METHOD Praca : BOOL
VAR_INPUT
END_VAR
tonOdczekaj (PT := REAL_TO_TIME (stParametry.rOdczekaj));
fbNaped.Praca ();

SUPER^.Praca ();
END_METHOD

METHOD Resetowanie : BOOL
VAR_INPUT
END_VAR
tonOdczekaj.IN								:= FALSE;

SUPER^.Resetowanie ();
END_METHOD

END_FUNCTION_BLOCK

// ---- POUs/93 - Podzespol/POU/FB_Podzespol.TcPOU
//==================================================================================================
//								RJM Maszyny sp. z o.o.
//									13.05.2022
//	Obsluga przesuwacza na siłowniku 
//	Siłownik zabieraka plus siłownik przesuwający 
//	Cykl przesuwania: wysun zabierak -> przesun -> schowaj zabierak -> powrót  
// 	v1.0	|| TC v 3.1.4024.22		|| - pierwsza wersja
//==================================================================================================
FUNCTION_BLOCK FB_Podzespol IMPLEMENTS ITF_Podzespol
VAR_INPUT
	//Parametry
END_VAR
VAR_OUTPUT
END_VAR
VAR
	//Elementy wejsciowe i wykonawcze
	bBazuj									: BOOL;
	bBazowanie								: BOOL;
	bCyklBazowaniaSkonczony					: BOOL;
	bPierwszePrzejscieBazowanie				: BOOL;
	iKrokBazowania							: INT :=0;

	bWykonajCyklPracy						: BOOL;
	bCyklPracy								: BOOL;
	bCyklPracySkonczony						: BOOL;
	bPierwszePrzejsciePracy					: BOOL;
	iKrokPracy								: INT := 0;

	bReset									: BOOL;
END_VAR

PROPERTY Bazowanie : BOOL
GET
Bazowanie									:= bBazowanie;
END_GET
END_PROPERTY

PROPERTY Bazuj : BOOL
SET
bBazuj										:= Bazuj;
END_SET
END_PROPERTY

METHOD CyklBazowania_Praca : BOOL
VAR_INPUT
END_VAR
END_METHOD

PROPERTY CyklPracy : BOOL
GET
CyklPracy								:= bCyklPracy;
END_GET
END_PROPERTY

METHOD CyklPracy_Praca : BOOL
VAR_INPUT
END_VAR
END_METHOD

PROPERTY CyklPracySkonczony : BOOL
GET
CyklPracySkonczony					:= bCyklPracySkonczony;
END_GET
END_PROPERTY

PROPERTY Pozycja0 : BOOL
GET
END_GET
END_PROPERTY

METHOD Praca : BOOL
VAR_INPUT
END_VAR
//---------------Resetowanie zmiennych
	IF (bReset) THEN
		Resetowanie ();
	END_IF
//---------------Resetowanie zmiennych
//---------------Bazowanie siłowników - powrót do poczatku
	IF (bBazuj) THEN
		bPierwszePrzejscieBazowanie				:= FALSE;
		bBazowanie								:= TRUE;
		bBazuj									:= FALSE;
	END_IF
	IF (bBazowanie) THEN
		bBazowanie								:= CyklBazowania_Praca ();
	END_IF
//---------------Bazowanie siłowników - powrót do poczatku
//---------------Cykl przesuwnaia - koniec gora dol poczatek
	IF (bWykonajCyklPracy) THEN
		bCyklPracy						:= TRUE;
	END_IF
	IF (bCyklPracy) THEN
		bCyklPracy						:= CyklPracy_Praca ();
	END_IF
//---------------Cykl przesuwnaia - koniec gora dol poczatek
END_METHOD

METHOD Resetowanie : BOOL
VAR_INPUT
END_VAR
bWykonajCyklPracy							:= FALSE;
bCyklPracy									:= FALSE;
bCyklPracySkonczony							:= FALSE;
bBazuj										:= false;
bBazowanie									:= false;
bCyklBazowaniaSkonczony						:= FALSE;
bPierwszePrzejscieBazowanie					:= FALSE;
bPierwszePrzejsciePracy						:= FALSE;
iKrokBazowania								:= 0;
iKrokPracy									:= 0;



bReset										:= FALSE;
END_METHOD

PROPERTY Resetuj : BOOL
SET
bReset										:=Resetuj;
END_SET
END_PROPERTY

PROPERTY WykonajCyklPracy : BOOL
SET
bWykonajCyklPracy						:= WykonajCyklPracy;
END_SET
END_PROPERTY

END_FUNCTION_BLOCK

// ---- POUs/03 - Ciecie/POU/FB_Ciecie_Komunikacja.TcPOU
FUNCTION_BLOCK FB_Ciecie_Komunikacja EXTENDS FB_LogowanieBledow_ElementZlozony
VAR_INPUT
END_VAR
VAR_OUTPUT
END_VAR
VAR
END_VAR

METHOD DefinicjaTabeliZdarzen_1031_Niemiecki : BOOL
VAR_INPUT
	arrTablicaDefinicjiZdarzenOpis			: REFERENCE TO ARRAY [1..GVL_LogowanieBledow_Stale.MAX_ILOSC_ZDARZEN] OF DUT_LogowanieBledow_ZdarzenieOpis;

END_VAR
//arrTablicaDefinicjiZdarzenOpis [iStartId+0].sOpis	:= 'DE - TESTOWA WIADOMOSC';
END_METHOD

METHOD DefinicjaTabeliZdarzen_1033_Angielski : BOOL
VAR_INPUT
	arrTablicaDefinicjiZdarzenOpis			: REFERENCE TO ARRAY [1..GVL_LogowanieBledow_Stale.MAX_ILOSC_ZDARZEN] OF DUT_LogowanieBledow_ZdarzenieOpis;

END_VAR
//arrTablicaDefinicjiZdarzenOpis [iStartId+0].sOpis	:= 'EN - TESTOWA WIADOMOSC';
END_METHOD

METHOD DefinicjaTabeliZdarzen_1045_Polski : BOOL
VAR_INPUT
	arrTablicaDefinicjiZdarzenOpis			: REFERENCE TO ARRAY [1..GVL_LogowanieBledow_Stale.MAX_ILOSC_ZDARZEN] OF DUT_LogowanieBledow_ZdarzenieOpis;

END_VAR
//arrTablicaDefinicjiZdarzenOpis [iStartId+0].sOpis	:= 'PL - TESTOWA WIADOMOSC';
END_METHOD

METHOD DefinicjaTabeliZdarzen_Ogolna : BOOL
VAR_INPUT
	arrTablicaDefinicjiZdarzen				: REFERENCE TO ARRAY [1..GVL_LogowanieBledow_Stale.MAX_ILOSC_ZDARZEN] OF DUT_LogowanieBledow_Zdarzenie;
	arrTablicaDefinicjiZdarzenOpis			: REFERENCE TO ARRAY [1..GVL_LogowanieBledow_Stale.MAX_ILOSC_ZDARZEN] OF DUT_LogowanieBledow_ZdarzenieOpis;
	arrTablicaDefinicjiZdarzenStan			: REFERENCE TO ARRAY [1..GVL_LogowanieBledow_Stale.MAX_ILOSC_ZDARZEN] OF DUT_LogowanieBledow_ZdarzenieStan;

	iIdZdarzenia							: REFERENCE TO INT;
	iNrPodzespolu							: INT := 0;
	iNrPodelementu							: INT := 0;
	iNrElementu								: INT := 0;
END_VAR
(*
//testowy blad
	iIdZdarzenia												:= iIdZdarzenia + 1;
	arrTablicaDefinicjiZdarzen [iIdZdarzenia].iIdZdarzenia		:= iIdZdarzenia;
	arrTablicaDefinicjiZdarzen [iIdZdarzenia].byRodzajZdarzenia	:= 3;
	arrTablicaDefinicjiZdarzen [iIdZdarzenia].sKodBledu			:= '0001';
	arrTablicaDefinicjiZdarzen [iIdZdarzenia].sNrKomponentu		:= GenerujNrKomponentu (iNrPodzespolu := iNrPodzespolu, iNrPodelementu := iNrPodelementu, iNrElementu := iNrElementu); 
	arrTablicaDefinicjiZdarzenOpis [iIdZdarzenia].iIdZdarzenia 	:= iIdZdarzenia;
	arrTablicaDefinicjiZdarzenStan [iIdZdarzenia].iIdZdarzenia 	:= iIdZdarzenia;
	arrTablicaDefinicjiZdarzenStan [iIdZdarzenia].bAktywne		:= FALSE;
	*)
END_METHOD

END_FUNCTION_BLOCK

// ---- POUs/95 - Logowanie bledow/POU/FB_LogowanieBledow_ElementZlozony.TcPOU
//==================================================================================================
//								RJM Maszyny sp. z o.o.
//									14.06.2022
//	FB posredniczący pomiędzy FB a logerem alarmów  rozszerzenie dla elementów złożonych
// 	v1.0	|| TC v 3.1.4024.22		|| - pierwsza wersja
//==================================================================================================
FUNCTION_BLOCK FB_LogowanieBledow_ElementZlozony EXTENDS FB_LogowanieBledow_ElementWykonawczy
VAR_INPUT
	
END_VAR
VAR_OUTPUT
END_VAR
VAR
	arrElementyWykonawcze 					: ARRAY [1..GVL_LogowanieBledow_Stale.MAX_ILOSC_ELEMENTOW_NA_PODZESPOL] OF ITF_LogowanieBledow_ElementWykonawczy;
	iIloscPodlementow						: INT;
END_VAR

METHOD DefinicjaTabeliZdarzen_1031_Niemiecki : BOOL
VAR_INPUT
	arrTablicaDefinicjiZdarzenOpis			: REFERENCE TO ARRAY [1..GVL_LogowanieBledow_Stale.MAX_ILOSC_ZDARZEN] OF DUT_LogowanieBledow_ZdarzenieOpis;

END_VAR
END_METHOD

METHOD DefinicjaTabeliZdarzen_1033_Angielski : BOOL
VAR_INPUT
	arrTablicaDefinicjiZdarzenOpis			: REFERENCE TO ARRAY [1..GVL_LogowanieBledow_Stale.MAX_ILOSC_ZDARZEN] OF DUT_LogowanieBledow_ZdarzenieOpis;

END_VAR
END_METHOD

METHOD DefinicjaTabeliZdarzen_1045_Polski : BOOL
VAR_INPUT
	arrTablicaDefinicjiZdarzenOpis			: REFERENCE TO ARRAY [1..GVL_LogowanieBledow_Stale.MAX_ILOSC_ZDARZEN] OF DUT_LogowanieBledow_ZdarzenieOpis;

END_VAR
END_METHOD

METHOD DefinicjaTabeliZdarzen_Ogolna : BOOL
VAR_INPUT
	arrTablicaDefinicjiZdarzen				: REFERENCE TO ARRAY [1..GVL_LogowanieBledow_Stale.MAX_ILOSC_ZDARZEN] OF DUT_LogowanieBledow_Zdarzenie;
	arrTablicaDefinicjiZdarzenOpis			: REFERENCE TO ARRAY [1..GVL_LogowanieBledow_Stale.MAX_ILOSC_ZDARZEN] OF DUT_LogowanieBledow_ZdarzenieOpis;
	arrTablicaDefinicjiZdarzenStan			: REFERENCE TO ARRAY [1..GVL_LogowanieBledow_Stale.MAX_ILOSC_ZDARZEN] OF DUT_LogowanieBledow_ZdarzenieStan;

	iIdZdarzenia							: REFERENCE TO INT;
	iNrPodzespolu							: INT := 0;
	iNrPodelementu							: INT := 0;
	iNrElementu								: INT := 0;
END_VAR
END_METHOD

METHOD FB_init : BOOL
VAR_INPUT
	bInitRetains : BOOL; // if TRUE, the retain variables are initialized (warm start / cold start)
	bInCopyCode : BOOL;  // if TRUE, the instance afterwards gets moved into the copy code (online change)
	arrElementyWykonawcze 					: ARRAY [1..10] OF ITF_LogowanieBledow_ElementWykonawczy;
	iIloscPodlementow						: INT;
END_VAR
THIS^.arrElementyWykonawcze					:= arrElementyWykonawcze;
THIS^.iIloscPodlementow						:= iIloscPodlementow;
END_METHOD

METHOD ZwrocTabliceDefinicji : BOOL
VAR_INPUT
	arrTablicaDefinicjiZdarzen				: REFERENCE TO ARRAY [1..GVL_LogowanieBledow_Stale.MAX_ILOSC_ZDARZEN] OF DUT_LogowanieBledow_Zdarzenie;
	arrTablicaDefinicjiZdarzenOpis			: REFERENCE TO ARRAY [1..GVL_LogowanieBledow_Stale.MAX_ILOSC_ZDARZEN] OF DUT_LogowanieBledow_ZdarzenieOpis;
	arrTablicaDefinicjiZdarzenStan			: REFERENCE TO ARRAY [1..GVL_LogowanieBledow_Stale.MAX_ILOSC_ZDARZEN] OF DUT_LogowanieBledow_ZdarzenieStan;
	
	iIdZdarzenia							: REFERENCE TO INT;
	iNrPodzespolu							: INT;
	iNrPodelementu							: INT;
	iNrElementu								: INT;
	iJezykId								: INT;
END_VAR
VAR
	iI: INT;
END_VAR
//Zwrócenie definicji zdarzen dla głównego elementu 
SUPER^.ZwrocTabliceDefinicji (	arrTablicaDefinicjiZdarzen := arrTablicaDefinicjiZdarzen,
								arrTablicaDefinicjiZdarzenOpis := arrTablicaDefinicjiZdarzenOpis,
								arrTablicaDefinicjiZdarzenStan := arrTablicaDefinicjiZdarzenStan,
								iIdZdarzenia := iIdZdarzenia,
								iNrPodzespolu := iNrPodzespolu, 
								iNrPodelementu := iNrPodelementu,
								iNrElementu := 1, 
								iJezykId := iJezykID);
//zwrócenie tablicy definicji dla podelementów

	FOR iI := 1 TO iIloscPodlementow DO 
		arrElementyWykonawcze [iI].ZwrocTabliceDefinicji (	arrTablicaDefinicjiZdarzen := arrTablicaDefinicjiZdarzen,
															arrTablicaDefinicjiZdarzenOpis := arrTablicaDefinicjiZdarzenOpis,
															arrTablicaDefinicjiZdarzenStan := arrTablicaDefinicjiZdarzenStan,
															iIdZdarzenia := iIdZdarzenia, 
															iNrPodzespolu := iNrPodzespolu, 
															iNrPodelementu := iNrPodelementu,
															iNrElementu := iI+1, 
															iJezykId := iJezykID);
	END_FOR
END_METHOD

METHOD ZwrocTabliceStanu : BOOL
VAR_INPUT
	arrTablicaDefinicjiZdarzenStan			: REFERENCE TO ARRAY [1..GVL_LogowanieBledow_Stale.MAX_ILOSC_ZDARZEN] OF DUT_LogowanieBledow_ZdarzenieStan;
END_VAR

VAR
	iI										: INT;
	iJ										: INT;
END_VAR
SUPER^.ZwrocTabliceStanu (arrTablicaDefinicjiZdarzenStan := arrTablicaDefinicjiZdarzenStan);

FOR iJ := 1 TO iIloscPodlementow DO
	arrElementyWykonawcze [iJ].ZwrocTabliceStanu (arrTablicaDefinicjiZdarzenStan := arrTablicaDefinicjiZdarzenStan);
END_FOR
END_METHOD

END_FUNCTION_BLOCK

// ---- POUs/02 - Przesuwacz Na Silowniku/POU/FB_PrzesuwaczNaSilowniku.TcPOU
//==================================================================================================
//								RJM Maszyny sp. z o.o.
//									13.05.2022
//	Obsluga przesuwacza na siłowniku 
//	Siłownik zabieraka plus siłownik przesuwający 
//	Cykl przesuwania: wysun zabierak -> przesun -> schowaj zabierak -> powrót  
// 	v1.0	|| TC v 3.1.4024.22		|| - pierwsza wersja
//==================================================================================================
FUNCTION_BLOCK FB_PrzesuwaczNaSilowniku EXTENDS FB_Podzespol
VAR_INPUT
	stParametry								: DUT_PrzesuwaczNaSilowniku_Parametry;
END_VAR
VAR_OUTPUT
END_VAR
VAR
	bCzujnik0Zabieraka						: ITF_Czujnik;
	bCzujnikMaxZabieraka					: ITF_Czujnik;
	fbElektrozaworZabieraka					: ITF_Elektozawor;
	bCzujnik0Przesuwacza					: ITF_Czujnik;
	bCzujnikMaxPrzesuwacza					: ITF_Czujnik;
	fbElektrozaworPrzesuwacza				: ITF_Elektozawor;
	fbZabierak								: FB_Silownik_Kontrola (	fbCzujnikPozycja0 			:= GVL_Wejscia_IO.bCzujnik0PW_Z, 
																		fbCzujnikPozycjaMax 		:= GVL_Wejscia_IO.bCzujnikMaxPW_Z,
																		fbElektrozawor 				:= GVL_Wyjscia_IO.fbElektrozaworPW_Z);
	fbPrzesuwanie							: FB_Silownik_Kontrola (	fbCzujnikPozycja0 			:= GVL_Wejscia_IO.bCzujnik0PW_N, 
																		fbCzujnikPozycjaMax 		:= GVL_Wejscia_IO.bCzujnikMaxPW_N,
																		fbElektrozawor 				:= GVL_Wyjscia_IO.fbElektrozaworPW_N);

	arrElementyWykonawcze 					: ARRAY [1..GVL_LogowanieBledow_Stale.MAX_ILOSC_ELEMENTOW_NA_PODZESPOL] OF ITF_LogowanieBledow_ElementWykonawczy := 
														[fbZabierak.fbLBKomunikacja, 
														fbPrzesuwanie.fbLBKomunikacja];
	fbLBKomunikacja							: FB_PrzesuwaczNaSilowniku_Komunikacja 
														(arrElementyWykonawcze := arrElementyWykonawcze,
														iIloscPodlementow := 2);

	tonChwilaPoDojechaniu					: TON;
END_VAR

METHOD CyklBazowania_Praca : BOOL
VAR_INPUT
END_VAR
IF (NOT bPierwszePrzejscieBazowanie) THEN
	bPierwszePrzejscieBazowanie				:= TRUE;
	bCyklBazowaniaSkonczony					:= FALSE;
	fbZabierak.PrzesunDoPoczatku			:= TRUE;
	iKrokBazowania							:= 1;
END_IF

CASE iKrokBazowania OF
	1	:
		IF (fbZabierak.NaPoczatku) THEN
			fbPrzesuwanie.PrzesunDoPoczatku	:= TRUE;
			iKrokBazowania					:= 10;
		END_IF
		CyklBazowania_Praca					:= TRUE;
	10	:
		IF (fbPrzesuwanie.NaPoczatku AND fbZabierak.NaPoczatku) THEN
			bPierwszePrzejscieBazowanie		:= FALSE;
			bCyklBazowaniaSkonczony			:= TRUE;
			CyklBazowania_Praca				:= FALSE;
			iKrokBazowania					:= 0;
		ELSE
			CyklBazowania_Praca				:= TRUE;
		END_IF
		
END_CASE
END_METHOD

METHOD CyklPracy_Praca : BOOL
VAR_INPUT
END_VAR
IF (NOT bPierwszePrzejsciePracy) THEN
	bPierwszePrzejsciePracy					:= TRUE;
	bCyklPracySkonczony						:= FALSE;
	fbZabierak.PrzesunDoKonca				:= TRUE;
	tonChwilaPoDojechaniu.IN				:= FALSE;
	iKrokPracy								:= 1;
END_IF

CASE iKrokPracy OF
	1	:
	IF (fbZabierak.NaKoncu) THEN
		fbPrzesuwanie.PrzesunDoKonca	:= TRUE;
		iKrokPracy							:= 10;
	END_IF
	CyklPracy_Praca							:= TRUE;
	10	:
	IF (fbPrzesuwanie.NaKoncu) THEN
		tonChwilaPoDojechaniu.IN			:= TRUE;
		iKrokPracy							:= 20;
	END_IF
	CyklPracy_Praca							:= TRUE;
	20	:
	IF (tonChwilaPoDojechaniu.Q) THEN
		tonChwilaPoDojechaniu.IN			:= FALSE;
		fbZabierak.PrzesunDoKonca			:= TRUE;
		iKrokPracy							:= 30;
	END_IF
	CyklPracy_Praca							:= TRUE;
	30	:
	IF (fbZabierak.NaPoczatku) THEN
		fbPrzesuwanie.PrzesunDoPoczatku	:= TRUE;
		iKrokPracy							:= 40;
	END_IF
	CyklPracy_Praca							:= TRUE;
	40	:
	IF (fbPrzesuwanie.NaPoczatku) THEN
		iKrokPracy							:= 50;
		bCyklPracySkonczony					:= TRUE;
	END_IF
	CyklPracy_Praca							:= TRUE;
	50	:
		iKrokPracy							:= 0;
		CyklPracy_Praca						:= FALSE;
END_CASE
END_METHOD

METHOD FB_init : BOOL
VAR_INPUT
	bInitRetains : BOOL; // if TRUE, the retain variables are initialized (warm start / cold start)
	bInCopyCode : BOOL;  // if TRUE, the instance afterwards gets moved into the copy code (online change)
	bCzujnik0Zabieraka						: ITF_Czujnik;
	bCzujnikMaxZabieraka					: ITF_Czujnik;
	fbElektrozaworZabieraka					: ITF_Elektozawor;
	bCzujnik0Przesuwacza					: ITF_Czujnik;
	bCzujnikMaxPrzesuwacza					: ITF_Czujnik;
	fbElektrozaworPrzesuwacza				: ITF_Elektozawor;
	
END_VAR

THIS^.bCzujnik0Zabieraka					:= bCzujnik0Zabieraka;			     
THIS^.bCzujnikMaxZabieraka					:= bCzujnikMaxZabieraka;		    
THIS^.fbElektrozaworZabieraka				:= fbElektrozaworZabieraka;		 
THIS^.bCzujnik0Przesuwacza					:= bCzujnik0Przesuwacza;		    
THIS^.bCzujnikMaxPrzesuwacza				:= bCzujnikMaxPrzesuwacza;		  
THIS^.fbElektrozaworPrzesuwacza				:= fbElektrozaworPrzesuwacza;

THIS^.fbZabierak.FB_init (FALSE, FALSE, bCzujnik0Zabieraka, bCzujnikMaxZabieraka, fbElektrozaworZabieraka);
THIS^.fbPrzesuwanie.FB_init (FALSE, FALSE, bCzujnik0Przesuwacza, bCzujnikMaxPrzesuwacza, fbElektrozaworPrzesuwacza);
END_METHOD

PROPERTY Pozycja0 : BOOL
GET
Pozycja0									:= fbZabierak.NaPoczatku AND fbPrzesuwanie.NaPoczatku;
END_GET
END_PROPERTY

METHOD Praca : BOOL
VAR_INPUT
END_VAR
tonChwilaPoDojechaniu (PT := REAL_TO_TIME (stParametry.rCzasNaKoncu));

fbZabierak.Praca ();
fbPrzesuwanie.Praca ();


SUPER^.Praca ();
END_METHOD

METHOD Resetowanie : BOOL
VAR_INPUT
END_VAR
tonChwilaPoDojechaniu.IN					:= FALSE;

SUPER^.Resetowanie ();
END_METHOD

END_FUNCTION_BLOCK

// ---- POUs/01 - Elementy/Czujnik/POU/FB_Czujnik_NO.TcPOU
//==================================================================================================
//								RJM Maszyny sp. z o.o.
//									04.06.2022
//	Obsługa czujnika  NO
// 	v1.0	|| TC v 3.1.4024.22		|| - pierwsza wersja
//==================================================================================================
FUNCTION_BLOCK FB_Czujnik_NO IMPLEMENTS ITF_Czujnik
VAR_INPUT
	bSymulacja								: BOOL;
END_VAR
VAR
	bWejscie						AT %I*	: BOOL;
END_VAR

//==================================================================================================
//								RJM Maszyny sp. z o.o.
//									13.05.2022
//	Informacja czy czujnik jest zadziałany 
// 	v1.0	|| TC v 3.1.4024.22		|| - pierwsza wersja
//==================================================================================================
PROPERTY CzyZadzialany : BOOL
GET
CzyZadzialany								:= bWejscie;
END_GET
END_PROPERTY

END_FUNCTION_BLOCK

// ---- POUs/01 - Elementy/Elektrozawór/POU/FB_Elektrozawor_5na2_2Cewki.TcPOU
//==================================================================================================
//								RJM Maszyny sp. z o.o.
//									04.06.2022
//	Sterowanie elektrozaworem  - 5 na 2 z dwiema cewkami
// 	v1.0	|| TC v 3.1.4024.22		|| - pierwsza wersja
//==================================================================================================
FUNCTION_BLOCK FB_Elektrozawor_5na2_2Cewki IMPLEMENTS ITF_Elektozawor
VAR
	bCewkaA							AT %Q*	: BOOL;		//Cewka sterująca wyjściem 2 - 0 do MAX
	bCewkaB							AT %Q*	: BOOL;		//Cewka sterująca wyjściem 4 - MAX do 0
END_VAR

(*==================================================================================================
								RJM Maszyny sp. z o.o.
									04.06.2022
	Sterowanie cewkami elektrozaworu 
 	v1.0	|| TC v 3.1.4024.22		|| - pierwsza wersja
==================================================================================================*)
METHOD Steruj : BOOL
VAR_INPUT
	bKierunekWstrone0						: BOOL;
	bKierunekWStroneMax						: BOOL;
END_VAR
IF (bKierunekWStroneMax AND NOT bCewkaA) THEN
	bCewkaA									:= TRUE;
END_IF
IF  (bKierunekWstrone0 AND bCewkaA) THEN
	bCewkaA									:= FALSE;
END_IF

IF (bKierunekWstrone0 AND NOT bCewkaB) THEN
	bCewkaB									:= TRUE;
END_IF
IF  (bKierunekWStroneMax AND bCewkaB) THEN
	bCewkaB									:= FALSE;
END_IF
END_METHOD

END_FUNCTION_BLOCK

// ---- POUs/90 - Stan Maszyny/POU/FB_StanMaszyny.TcPOU
//==================================================================================================
//								RJM Maszyny sp. z o.o.
//									13.05.2022
//	Sterowanie pracą maszyny i jej trybami  
// 	v1.0	|| TC v 3.1.4024.29		|| - pierwsza wersja
//==================================================================================================
FUNCTION_BLOCK FB_StanMaszyny
VAR_INPUT
	bStart                                  : BOOL;
	bStop                                   : bool;
	bReset                                  : bool;
	bAbort                                  : bool;
	bClear                                  : bool;
	bHold                                   : bool;
	bUnHold                                 : bool;
	bSuspend                                : bool;
	bUnsuspend								: BOOL;
	eTryb									: E_PMLUnitMode;	//zadany tryb pracy
END_VAR
VAR_OUTPUT
END_VAR
VAR
	arrVisuStany							: ARRAY [0..17] OF DUT_StanMaszyny_VISU_Stan;
	arrVisuTryb								: ARRAY [0..9] of ARRAY [0..17] OF BOOL;
	eStan									: E_PMLState := E_PMLState.ABORTING;		//aktualny stan maszyny
	eTrybPracy								: E_PMLUnitMode := E_PMLUnitMode.MANUAL;	//aktualny tryb pracy
	
	arrPodzesoly							: ARRAY [1..GVL_StanMaszyny_Stale.MAX_LICZBA_PODZESPOLOW] OF ITF_StanMaszyny;
	iIloscDodanychPodzespolow				: INT;

	iAktualnyStan							: INT;
	iPoprzedniStan							: INT;
	iNumerTrybuPracy						: INT;
	iPoprzedniTrybPracy						: INT;

	bResetingSkonczone						: BOOL;
	bStoppingZakonczone						: BOOL;
	bAbortingZakonczone						: BOOL;
	bClearingZakonczone						: BOOL;
	bCompletingZakonczone					: BOOL;
	bHoldingZakonczone						: BOOL;
	bStartingZakonczone						: BOOL;
	bSuspendingZakonczone					: BOOL;
	bUnholdingZakonczone					: BOOL;
	bUnsuspendingZakonczone					: BOOL;	
	bInicjalizacja							: BOOL;
	bPierwszePrzejscieWOperacji				: BOOL;
	arrOperacjaWykonana						: ARRAY [1..GVL_StanMaszyny_Stale.MAX_LICZBA_PODZESPOLOW] OF BOOL;	//tablica zakonczenia zadanej operacji przez podzespoly
END_VAR

IF (NOT bInicjalizacja) THEN
	bInicjalizacja							:= TRUE;
	Inicjalizacja ();
END_IF



StanMaszyny ();

METHOD FB_init : BOOL
VAR_INPUT
	bInitRetains : BOOL; // if TRUE, the retain variables are initialized (warm start / cold start)
	bInCopyCode : BOOL;  // if TRUE, the instance afterwards gets moved into the copy code (online change)
	arrPodzesoly							: ARRAY [1..GVL_StanMaszyny_Stale.MAX_LICZBA_PODZESPOLOW] OF ITF_StanMaszyny;
	iIloscDodanychPodzespolow				: INT;
END_VAR
THIS^.arrPodzesoly								:= arrPodzesoly;
THIS^.iIloscDodanychPodzespolow					:= iIloscDodanychPodzespolow;
END_METHOD

//==================================================================================================
//								RJM Maszyny sp. z o.o.
//									13.05.2022
//	Iniecjalizacja tablicy potrzebnej do wyświetlania diagramu  
// 	v1.0	|| TC v 3.1.4024.29		|| - pierwsza wersja
//==================================================================================================
METHOD PRIVATE Inicjalizacja : BOOL
VAR_INPUT
END_VAR

VAR
	i,j: INT;
END_VAR


FOR j := 0 TO 9 DO
	FOR i := 0 TO 17 DO
		arrVisuStany [i].bAktywny				:= FALSE;
		CASE i OF
			0	:
				arrVisuStany [i].sNazwa			:= 'UNDEFINED';
				arrVisuStany [i].dwKolorTla		:= 16#FFFF0000;	//czerwony
			1	:             
				arrVisuStany [i].sNazwa			:= 'CLEARING';
				arrVisuStany [i].dwKolorTla		:= 16#FF00FF00;	//zielony
			2	:             
				arrVisuStany [i].sNazwa			:= 'STOPPED';
				arrVisuStany [i].dwKolorTla		:= 16#FFFFFF00;	//zolty
			3	:
				arrVisuStany [i].sNazwa			:= 'STARTING';
				arrVisuStany [i].dwKolorTla		:= 16#FF00FF00;
			4	:             
				arrVisuStany [i].sNazwa			:= 'IDLE';
				arrVisuStany [i].dwKolorTla		:= 16#FFFFFF00;
			5	:             
				arrVisuStany [i].sNazwa			:= 'SUSPENDED';
				arrVisuStany [i].dwKolorTla		:= 16#FFFFFF00;		
			6	:             
				arrVisuStany [i].sNazwa			:= 'EXECUTE';
				arrVisuStany [i].dwKolorTla		:= 16#FF0000FF;
			7	:             
				arrVisuStany [i].sNazwa			:= 'STOPPING';
				arrVisuStany [i].dwKolorTla		:= 16#FF00FF00;
			8	:             
				arrVisuStany [i].sNazwa			:= 'ABORTING';
				arrVisuStany [i].dwKolorTla		:= 16#FF00FF00;		
			9	:             
				arrVisuStany [i].sNazwa			:= 'ABORTED';
				arrVisuStany [i].dwKolorTla		:= 16#FFFFFF00;
			10	:             
				arrVisuStany [i].sNazwa			:= 'HOLDING';
				arrVisuStany [i].dwKolorTla		:= 16#FF00FF00;
			11	:             
				arrVisuStany [i].sNazwa			:= 'HELD';
				arrVisuStany [i].dwKolorTla		:= 16#FFFFFF00;	
			12	:             
				arrVisuStany [i].sNazwa			:= 'UNHOLDING';
				arrVisuStany [i].dwKolorTla		:= 16#FF00FF00;
			13	:
				arrVisuStany [i].sNazwa			:= 'SUSPENDING';
				arrVisuStany [i].dwKolorTla		:= 16#FF00FF00;
			14	:             
				arrVisuStany [i].sNazwa			:= 'UNSUSPENDING';
				arrVisuStany [i].dwKolorTla		:= 16#FF00FF00;		
			15	:             
				arrVisuStany [i].sNazwa			:= 'RESETTING';
				arrVisuStany [i].dwKolorTla		:= 16#FF00FF00;
			16	:             
				arrVisuStany [i].sNazwa			:= 'COMPLETING';
				arrVisuStany [i].dwKolorTla		:= 16#FF00FF00;
			17	:             
				arrVisuStany [i].sNazwa			:= 'COMPLETE';
				arrVisuStany [i].dwKolorTla		:= 16#FFFFFF00;		
		END_CASE
	END_FOR
END_FOR
END_METHOD

//==================================================================================================
//								RJM Maszyny sp. z o.o.
//									13.05.2022
//	Konfiguracja który stan w jakim trybie ma być aktywny
// 	v1.0	|| TC v 3.1.4024.29		|| - pierwsza wersja
//==================================================================================================
METHOD KonfiguracjaStanowPracyDlaTrybu : BOOL
VAR_INPUT
	eNrTrybu								: E_PMLUnitMode;
	bClearing 								: BOOL;  
	bStopped 								: BOOL;  
	bStarting 								: BOOL;  
	bIdle 									: BOOL;  
	bSuspended 								: BOOL;  
	bExecute 								: BOOL;  
	bStopping	 							: BOOL;  
	bAborting 								: BOOL;  
	bAborted 								: BOOL;  
	bHolding 								: BOOL;  
	bHeld 									: BOOL;  
	bUnholding 								: BOOL;  
	bSuspending 							: BOOL;  
	bUnsuspending 							: BOOL;  
	bResetting 								: BOOL;  
	bCompleting 							: BOOL;  
	bComplete	 							: BOOL;  
END_VAR
CASE eNrTrybu OF
	E_PMLUnitMode.UNDEFINED		:
		arrVisuTryb [0][0] 						:= FALSE;						 
		arrVisuTryb [0][1] 						:= FALSE;						 
		arrVisuTryb [0][2] 						:= FALSE;						 
		arrVisuTryb [0][3] 						:= FALSE;						 
		arrVisuTryb [0][4] 						:= FALSE;						 
		arrVisuTryb [0][5] 						:= FALSE;						 
		arrVisuTryb [0][6] 						:= FALSE;						 
		arrVisuTryb [0][7] 						:= FALSE;						 
		arrVisuTryb [0][8] 						:= FALSE;						 
		arrVisuTryb [0][9] 						:= FALSE;						 
		arrVisuTryb [0][10] 					:= FALSE;						 
		arrVisuTryb [0][11] 					:= FALSE;						 
		arrVisuTryb [0][12] 					:= FALSE;						 
		arrVisuTryb [0][13] 					:= FALSE;						 
		arrVisuTryb [0][14] 					:= FALSE;						 
		arrVisuTryb [0][15] 					:= FALSE;						 
		arrVisuTryb [0][16] 					:= FALSE;						 
		arrVisuTryb [0][17] 					:= FALSE;						 	
	E_PMLUnitMode.AUTOMATIC		:
		arrVisuTryb [1][0] 						:= FALSE;								 
		arrVisuTryb [1][1] 						:= bClearing; 								 
		arrVisuTryb [1][2] 						:= bStopped; 								 
		arrVisuTryb [1][3] 						:= bStarting; 								 
		arrVisuTryb [1][4] 						:= bIdle; 									 
		arrVisuTryb [1][5] 						:= bSuspended; 								 
		arrVisuTryb [1][6] 						:= bExecute; 								 
		arrVisuTryb [1][7] 						:= bStopping;	 							 
		arrVisuTryb [1][8] 						:= bAborting; 								 
		arrVisuTryb [1][9] 						:= bAborted; 								 
		arrVisuTryb [1][10] 					:= bHolding; 								 
		arrVisuTryb [1][11] 					:= bHeld; 									 
		arrVisuTryb [1][12] 					:= bUnholding; 								 
		arrVisuTryb [1][13] 					:= bSuspending; 							 
		arrVisuTryb [1][14] 					:= bUnsuspending; 							 
		arrVisuTryb [1][15] 					:= bResetting;								 
		arrVisuTryb [1][16] 					:= bCompleting; 							 
		arrVisuTryb [1][17] 					:= bComplete;
	E_PMLUnitMode.MAINTENANCE 	:
		arrVisuTryb [2][0] 						:= FALSE;								 
		arrVisuTryb [2][1] 						:= bClearing; 								 
		arrVisuTryb [2][2] 						:= bStopped; 								 
		arrVisuTryb [2][3] 						:= bStarting; 								 
		arrVisuTryb [2][4] 						:= bIdle; 									 
		arrVisuTryb [2][5] 						:= bSuspended; 								 
		arrVisuTryb [2][6] 						:= bExecute; 								 
		arrVisuTryb [2][7] 						:= bStopping;	 							 
		arrVisuTryb [2][8] 						:= bAborting; 								 
		arrVisuTryb [2][9] 						:= bAborted; 								 
		arrVisuTryb [2][10] 					:= bHolding; 								 
		arrVisuTryb [2][11] 					:= bHeld; 									 
		arrVisuTryb [2][12] 					:= bUnholding; 								 
		arrVisuTryb [2][13] 					:= bSuspending; 							 
		arrVisuTryb [2][14] 					:= bUnsuspending; 							 
		arrVisuTryb [2][15] 					:= bResetting;								 
		arrVisuTryb [2][16] 					:= bCompleting; 							 
		arrVisuTryb [2][17] 					:= bComplete;
	E_PMLUnitMode.MANUAL 		:
		arrVisuTryb [3][0] 						:= FALSE;								 
		arrVisuTryb [3][1] 						:= bClearing; 								 
		arrVisuTryb [3][2] 						:= bStopped; 								 
		arrVisuTryb [3][3] 						:= bStarting; 								 
		arrVisuTryb [3][4] 						:= bIdle; 									 
		arrVisuTryb [3][5] 						:= bSuspended; 								 
		arrVisuTryb [3][6] 						:= bExecute; 								 
		arrVisuTryb [3][7] 						:= bStopping;	 							 
		arrVisuTryb [3][8] 						:= bAborting; 								 
		arrVisuTryb [3][9] 						:= bAborted; 								 
		arrVisuTryb [3][10] 					:= bHolding; 								 
		arrVisuTryb [3][11] 					:= bHeld; 									 
		arrVisuTryb [3][12] 					:= bUnholding; 								 
		arrVisuTryb [3][13] 					:= bSuspending; 							 
		arrVisuTryb [3][14] 					:= bUnsuspending; 							 
		arrVisuTryb [3][15] 					:= bResetting;								 
		arrVisuTryb [3][16] 					:= bCompleting; 							 
		arrVisuTryb [3][17] 					:= bComplete;
	E_PMLUnitMode.SEMIAUTOMATIC	:
		arrVisuTryb [4][0] 						:= FALSE;								 
		arrVisuTryb [4][1] 						:= bClearing; 								 
		arrVisuTryb [4][2] 						:= bStopped; 								 
		arrVisuTryb [4][3] 						:= bStarting; 								 
		arrVisuTryb [4][4] 						:= bIdle; 									 
		arrVisuTryb [4][5] 						:= bSuspended; 								 
		arrVisuTryb [4][6] 						:= bExecute; 								 
		arrVisuTryb [4][7] 						:= bStopping;	 							 
		arrVisuTryb [4][8] 						:= bAborting; 								 
		arrVisuTryb [4][9] 						:= bAborted; 								 
		arrVisuTryb [4][10] 					:= bHolding; 								 
		arrVisuTryb [4][11] 					:= bHeld; 									 
		arrVisuTryb [4][12] 					:= bUnholding; 								 
		arrVisuTryb [4][13] 					:= bSuspending; 							 
		arrVisuTryb [4][14] 					:= bUnsuspending; 							 
		arrVisuTryb [4][15] 					:= bResetting;								 
		arrVisuTryb [4][16] 					:= bCompleting; 							 
		arrVisuTryb [4][17] 					:= bComplete;
	E_PMLUnitMode.DRYRUN		:
		arrVisuTryb [5][0] 						:= FALSE;								 
		arrVisuTryb [5][1] 						:= bClearing; 								 
		arrVisuTryb [5][2] 						:= bStopped; 								 
		arrVisuTryb [5][3] 						:= bStarting; 								 
		arrVisuTryb [5][4] 						:= bIdle; 									 
		arrVisuTryb [5][5] 						:= bSuspended; 								 
		arrVisuTryb [5][6] 						:= bExecute; 								 
		arrVisuTryb [5][7] 						:= bStopping;	 							 
		arrVisuTryb [5][8] 						:= bAborting; 								 
		arrVisuTryb [5][9] 						:= bAborted; 								 
		arrVisuTryb [5][10] 					:= bHolding; 								 
		arrVisuTryb [5][11] 					:= bHeld; 									 
		arrVisuTryb [5][12] 					:= bUnholding; 								 
		arrVisuTryb [5][13] 					:= bSuspending; 							 
		arrVisuTryb [5][14] 					:= bUnsuspending; 							 
		arrVisuTryb [5][15] 					:= bResetting;								 
		arrVisuTryb [5][16] 					:= bCompleting; 							 
		arrVisuTryb [5][17] 					:= bComplete;
	E_PMLUnitMode.USERMODE1		:
		arrVisuTryb [6][0] 						:= FALSE;								 
		arrVisuTryb [6][1] 						:= bClearing; 								 
		arrVisuTryb [6][2] 						:= bStopped; 								 
		arrVisuTryb [6][3] 						:= bStarting; 								 
		arrVisuTryb [6][4] 						:= bIdle; 									 
		arrVisuTryb [6][5] 						:= bSuspended; 								 
		arrVisuTryb [6][6] 						:= bExecute; 								 
		arrVisuTryb [6][7] 						:= bStopping;	 							 
		arrVisuTryb [6][8] 						:= bAborting; 								 
		arrVisuTryb [6][9] 						:= bAborted; 								 
		arrVisuTryb [6][10] 					:= bHolding; 								 
		arrVisuTryb [6][11] 					:= bHeld; 									 
		arrVisuTryb [6][12] 					:= bUnholding; 								 
		arrVisuTryb [6][13] 					:= bSuspending; 							 
		arrVisuTryb [6][14] 					:= bUnsuspending; 							 
		arrVisuTryb [6][15] 					:= bResetting;								 
		arrVisuTryb [6][16] 					:= bCompleting; 							 
		arrVisuTryb [6][17] 					:= bComplete;
	E_PMLUnitMode.USERMODE2		:
		arrVisuTryb [7][0] 						:= FALSE;								 
		arrVisuTryb [7][1] 						:= bClearing; 								 
		arrVisuTryb [7][2] 						:= bStopped; 								 
		arrVisuTryb [7][3] 						:= bStarting; 								 
		arrVisuTryb [7][4] 						:= bIdle; 									 
		arrVisuTryb [7][5] 						:= bSuspended; 								 
		arrVisuTryb [7][6] 						:= bExecute; 								 
		arrVisuTryb [7][7] 						:= bStopping;	 							 
		arrVisuTryb [7][8] 						:= bAborting; 								 
		arrVisuTryb [7][9] 						:= bAborted; 								 
		arrVisuTryb [7][10] 					:= bHolding; 								 
		arrVisuTryb [7][11] 					:= bHeld; 									 
		arrVisuTryb [7][12] 					:= bUnholding; 								 
		arrVisuTryb [7][13] 					:= bSuspending; 							 
		arrVisuTryb [7][14] 					:= bUnsuspending; 							 
		arrVisuTryb [7][15] 					:= bResetting;								 
		arrVisuTryb [7][16] 					:= bCompleting; 							 
		arrVisuTryb [7][17] 					:= bComplete;
	E_PMLUnitMode.IDLE 			:
		arrVisuTryb [8][0] 						:= FALSE;								 
		arrVisuTryb [8][1] 						:= bClearing; 								 
		arrVisuTryb [8][2] 						:= bStopped; 								 
		arrVisuTryb [8][3] 						:= bStarting; 								 
		arrVisuTryb [8][4] 						:= bIdle; 									 
		arrVisuTryb [8][5] 						:= bSuspended; 								 
		arrVisuTryb [8][6] 						:= bExecute; 								 
		arrVisuTryb [8][7] 						:= bStopping;	 							 
		arrVisuTryb [8][8] 						:= bAborting; 								 
		arrVisuTryb [8][9] 						:= bAborted; 								 
		arrVisuTryb [8][10] 					:= bHolding; 								 
		arrVisuTryb [8][11] 					:= bHeld; 									 
		arrVisuTryb [8][12] 					:= bUnholding; 								 
		arrVisuTryb [8][13] 					:= bSuspending; 							 
		arrVisuTryb [8][14] 					:= bUnsuspending; 							 
		arrVisuTryb [8][15] 					:= bResetting;								 
		arrVisuTryb [8][16] 					:= bCompleting; 							 
		arrVisuTryb [8][17] 					:= bComplete;
	E_PMLUnitMode.ESTOP 		:
		arrVisuTryb [9][0] 						:= FALSE;								 
		arrVisuTryb [9][1] 						:= bClearing; 								 
		arrVisuTryb [9][2] 						:= bStopped; 								 
		arrVisuTryb [9][3] 						:= bStarting; 								 
		arrVisuTryb [9][4] 						:= bIdle; 									 
		arrVisuTryb [9][5] 						:= bSuspended; 								 
		arrVisuTryb [9][6] 						:= bExecute; 								 
		arrVisuTryb [9][7] 						:= bStopping;	 							 
		arrVisuTryb [9][8] 						:= bAborting; 								 
		arrVisuTryb [9][9] 						:= bAborted; 								 
		arrVisuTryb [9][10] 					:= bHolding; 								 
		arrVisuTryb [9][11] 					:= bHeld; 									 
		arrVisuTryb [9][12] 					:= bUnholding; 								 
		arrVisuTryb [9][13] 					:= bSuspending; 							 
		arrVisuTryb [9][14] 					:= bUnsuspending; 							 
		arrVisuTryb [9][15] 					:= bResetting;								 
		arrVisuTryb [9][16] 					:= bCompleting; 							 
		arrVisuTryb [9][17] 					:= bComplete;
END_CASE
END_METHOD

//==================================================================================================
//								RJM Maszyny sp. z o.o.
//									13.05.2022
//	Metodwa pomocnicza   
// 	v1.0	|| TC v 3.1.4024.29		|| - pierwsza wersja
//==================================================================================================
METHOD PRIVATE NacisnietyAbortPrzejscieDoAborting : BOOL
VAR_INPUT
END_VAR
	bResetingSkonczone						:= FALSE;	
	bStoppingZakonczone						:= FALSE;
	bAbortingZakonczone						:= FALSE;
	bClearingZakonczone						:= FALSE;
	bCompletingZakonczone					:= FALSE;
	bHoldingZakonczone						:= FALSE;
	bStartingZakonczone						:= FALSE;
	bSuspendingZakonczone					:= FALSE;
	bUnholdingZakonczone					:= FALSE;
	bUnsuspendingZakonczone					:= FALSE;
	bPierwszePrzejscieWOperacji				:= FALSE;
	eStan									:= E_PMLState.ABORTING;
END_METHOD

//==================================================================================================
//								RJM Maszyny sp. z o.o.
//									13.05.2022
//	Metoda pomocnicza 
// 	v1.0	|| TC v 3.1.4024.29		|| - pierwsza wersja
//==================================================================================================
METHOD PRIVATE NacisnietyStopPrzejscieDoStopping : BOOL
VAR_INPUT
END_VAR
	bResetingSkonczone						:= FALSE;	
	bStoppingZakonczone						:= FALSE;
	bAbortingZakonczone						:= FALSE;
	bClearingZakonczone						:= FALSE;
	bCompletingZakonczone					:= FALSE;
	bHoldingZakonczone						:= FALSE;
	bStartingZakonczone						:= FALSE;
	bSuspendingZakonczone					:= FALSE;
	bUnholdingZakonczone					:= FALSE;
	bUnsuspendingZakonczone					:= FALSE;
	bPierwszePrzejscieWOperacji				:= FALSE;
	eStan									:= E_PMLState.STOPPING;
END_METHOD

//==================================================================================================
//								RJM Maszyny sp. z o.o.
//									13.05.2022
//	Obsługa stanu ABORTED  
// 	v1.0	|| TC v 3.1.4024.29		|| - pierwsza wersja
//==================================================================================================
METHOD SM_Aborted : BOOL
VAR_INPUT
END_VAR

VAR
	i: INT;
END_VAR
FOR i := 1 TO iIloscDodanychPodzespolow DO
	arrPodzesoly [i].SM_Aborted ();
END_FOR

IF (bClear) THEN
	eStan									:= E_PMLState.CLEARING;
ELSIF (bStop) THEN
	eStan									:= E_PMLState.STOPPING;
ELSIF (bAbort) THEN
	eStan									:= E_PMLState.ABORTING;	
END_IF
//ZMIANA TRYBU PRACY
IF (eTryb <> eTrybPracy) THEN
//	IF (iNumerTrybuPracy <>iPoprzedniTrybPracy) THEN
		eTrybPracy								:= eTryb;
		iPoprzedniTrybPracy						:= iNumerTrybuPracy;
		eStan									:= E_PMLState.ABORTING;
//	END_IF
END_IF
//ZMIANA TRYBU PRACY
END_METHOD

//==================================================================================================
//								RJM Maszyny sp. z o.o.
//									13.05.2022
//	Obsługa stanu ABORTING
// 	v1.0	|| TC v 3.1.4024.29		|| - pierwsza wersja
//==================================================================================================
METHOD SM_Aborting : BOOL
VAR_INPUT
END_VAR

VAR
	i										: INT;
	bAbortingOK								: BOOL := TRUE;
END_VAR
IF (NOT bPierwszePrzejscieWOperacji) THEN
	FOR i := 1 TO iIloscDodanychPodzespolow DO
		arrOperacjaWykonana [i] 			:= FALSE;
	END_FOR
	bPierwszePrzejscieWOperacji				:= TRUE;
END_IF
FOR i := 1 TO iIloscDodanychPodzespolow DO
	IF (NOT arrOperacjaWykonana [i]) THEN
		arrOperacjaWykonana [i]				:= arrPodzesoly [i].SM_Aborting ();
	END_IF
	bAbortingOK								:= bAbortingOK AND arrOperacjaWykonana [i];
END_FOR

IF (bAbortingZakonczone OR bAbortingOK) THEN
	bAbortingZakonczone						:= FALSE;
	bPierwszePrzejscieWOperacji				:= FALSE;
	eStan									:= E_PMLState.ABORTED;
//ELSIF (bStop) THEN
//	eStan									:= E_PMLState.STOPPING;
//ELSIF (bAbort) THEN
//	eStan									:= E_PMLState.ABORTING;
END_IF
END_METHOD

//==================================================================================================
//								RJM Maszyny sp. z o.o.
//									13.05.2022
//	Obsługa stanu CLEARING  
// 	v1.0	|| TC v 3.1.4024.29		|| - pierwsza wersja
//==================================================================================================
METHOD SM_Clearing : BOOL
VAR_INPUT
END_VAR

VAR
	i										: INT;
	bClearingOK								: BOOL := TRUE;
END_VAR
IF (NOT bPierwszePrzejscieWOperacji) THEN
	FOR i := 1 TO iIloscDodanychPodzespolow DO
		arrOperacjaWykonana [i] 			:= FALSE;
	END_FOR
	bPierwszePrzejscieWOperacji				:= TRUE;
END_IF
FOR i := 1 TO iIloscDodanychPodzespolow DO
	IF (NOT arrOperacjaWykonana [i]) THEN
		arrOperacjaWykonana [i]				:= arrPodzesoly [i].SM_Clearing ();
	END_IF
	bClearingOK								:= bClearingOK AND arrOperacjaWykonana [i];
END_FOR

IF (bClearingZakonczone OR bClearingOK) THEN
	bClearingZakonczone						:= FALSE;
	bPierwszePrzejscieWOperacji				:= FALSE;
	eStan									:= E_PMLState.STOPPED;
END_IF
END_METHOD

//==================================================================================================
//								RJM Maszyny sp. z o.o.
//									13.05.2022
//	Obsługa stanu COMPLETE  
// 	v1.0	|| TC v 3.1.4024.29		|| - pierwsza wersja
//==================================================================================================
METHOD SM_Complete : BOOL
VAR_INPUT
END_VAR

VAR
	i: INT;
END_VAR
FOR i := 1 TO iIloscDodanychPodzespolow DO
	arrPodzesoly [i].SM_Complete ();
END_FOR

IF (bReset) THEN
	eStan									:= E_PMLState.RESETTING;
ELSIF (bStop) THEN
	NacisnietyStopPrzejscieDoStopping ();
ELSIF (bAbort) THEN
	NacisnietyAbortPrzejscieDoAborting ();
END_IF
END_METHOD

//==================================================================================================
//								RJM Maszyny sp. z o.o.
//									13.05.2022
//	Obsługa stanu COMPLITING  
// 	v1.0	|| TC v 3.1.4024.29		|| - pierwsza wersja
//==================================================================================================
METHOD SM_Completing : BOOL
VAR_INPUT
END_VAR

VAR
	i										: INT;
	bCompletingOK							: BOOL := TRUE;
END_VAR
IF (NOT bPierwszePrzejscieWOperacji) THEN
	FOR i := 1 TO iIloscDodanychPodzespolow DO
		arrOperacjaWykonana [i] 			:= FALSE;
	END_FOR
	bPierwszePrzejscieWOperacji				:= TRUE;
END_IF
FOR i := 1 TO iIloscDodanychPodzespolow DO
	IF (NOT arrOperacjaWykonana [i]) THEN
		arrOperacjaWykonana [i]					:= arrPodzesoly [i].SM_Completing ();
	END_IF
	bCompletingOK								:= bCompletingOK AND arrOperacjaWykonana [i];
END_FOR

IF (bCompletingZakonczone OR bCompletingOK) THEN
	eStan									:= E_PMLState.COMPLETE;
	bCompletingZakonczone					:= FALSE;
	bPierwszePrzejscieWOperacji				:= FALSE;
ELSIF (bStop) THEN
	NacisnietyStopPrzejscieDoStopping ();
ELSIF (bAbort) THEN
	NacisnietyAbortPrzejscieDoAborting ();
END_IF
END_METHOD

//==================================================================================================
//								RJM Maszyny sp. z o.o.
//									13.05.2022
//	Obsługa stanu EXECUTE  
// 	v1.0	|| TC v 3.1.4024.29		|| - pierwsza wersja
//==================================================================================================
METHOD SM_Execute : BOOL
VAR_INPUT
	eTrybPracy								: E_PMLUnitMode;
END_VAR
VAR
	i										: INT;
END_VAR
FOR i := 1 TO iIloscDodanychPodzespolow DO
	arrPodzesoly [i].SM_Execute (eTrybPracy := eTrybPracy);
END_FOR

IF (bHold) THEN
	eStan									:= E_PMLState.HOLDING;
ELSIF (bSuspend) THEN
	eStan									:= E_PMLState.SUSPENDING;
ELSIF (bStop) THEN
	NacisnietyStopPrzejscieDoStopping ();
ELSIF (bAbort) THEN
	NacisnietyAbortPrzejscieDoAborting ();
END_IF
END_METHOD

//==================================================================================================
//								RJM Maszyny sp. z o.o.
//									13.05.2022
//	Obsługa stanu HELD  
// 	v1.0	|| TC v 3.1.4024.29		|| - pierwsza wersja
//==================================================================================================
METHOD SM_Held : BOOL
VAR_INPUT
END_VAR

VAR
	i: INT;
END_VAR
FOR i := 1 TO iIloscDodanychPodzespolow DO
	arrPodzesoly [i].SM_Held ();
END_FOR

IF (bUnHold) THEN
	eStan									:= E_PMLState.UNHOLDING;
ELSIF (bStop) THEN
	NacisnietyStopPrzejscieDoStopping ();
ELSIF (bAbort) THEN
	NacisnietyAbortPrzejscieDoAborting ();
END_IF
END_METHOD

//==================================================================================================
//								RJM Maszyny sp. z o.o.
//									13.05.2022
//	Obsługa stanu HOLDING - wsztrymanie pracy przez maszyne  
// 	v1.0	|| TC v 3.1.4024.29		|| - pierwsza wersja
//==================================================================================================
METHOD SM_Holding : BOOL
VAR_INPUT
END_VAR

VAR
	i										: INT;
	bHoldingOK								: BOOL := TRUE;
END_VAR
IF (NOT bPierwszePrzejscieWOperacji) THEN
	FOR i := 1 TO iIloscDodanychPodzespolow DO
		arrOperacjaWykonana [i] 			:= FALSE;
	END_FOR
	bPierwszePrzejscieWOperacji				:= TRUE;
END_IF
FOR i := 1 TO iIloscDodanychPodzespolow DO
	IF (NOT arrOperacjaWykonana [i]) THEN
		arrOperacjaWykonana [i]				:= arrPodzesoly [i].SM_Holding ();
	END_IF
	bHoldingOK								:= bHoldingOK AND arrOperacjaWykonana [i];
END_FOR

IF (bHoldingZakonczone OR bHoldingOK) THEN
	bHoldingZakonczone						:= FALSE;
	bPierwszePrzejscieWOperacji				:= FALSE;
	eStan									:= E_PMLState.HELD;
ELSIF (bStop) THEN
	NacisnietyStopPrzejscieDoStopping ();
ELSIF (bAbort) THEN
	NacisnietyAbortPrzejscieDoAborting ();
END_IF
END_METHOD

//==================================================================================================
//								RJM Maszyny sp. z o.o.
//									13.05.2022
//	Obsługa stanu IDLE - maszyna gotowado pracy  
// 	v1.0	|| TC v 3.1.4024.29		|| - pierwsza wersja
//==================================================================================================
METHOD SM_Idle : BOOL
VAR_INPUT
END_VAR

VAR
	i: INT;
END_VAR
FOR i := 1 TO iIloscDodanychPodzespolow DO
	arrPodzesoly [i].SM_Idle ();
END_FOR

IF (bStart) THEN
	eStan									:= E_PMLState.STARTING;
ELSIF (bStop) THEN
	NacisnietyStopPrzejscieDoStopping ();
ELSIF (bAbort) THEN
	NacisnietyAbortPrzejscieDoAborting ();
END_IF
END_METHOD

//==================================================================================================
//								RJM Maszyny sp. z o.o.
//									13.05.2022
//	Obsługa stanu RESETTING  
// 	v1.0	|| TC v 3.1.4024.29		|| - pierwsza wersja
//==================================================================================================
METHOD SM_Resetting : BOOL
VAR_INPUT
END_VAR
VAR
	i										: INT;
	bResetingOK								: BOOL := TRUE;
END_VAR
IF (NOT bPierwszePrzejscieWOperacji) THEN
	FOR i := 1 TO iIloscDodanychPodzespolow DO
		arrOperacjaWykonana [i] 			:= FALSE;
	END_FOR
	bPierwszePrzejscieWOperacji				:= TRUE;
END_IF
FOR i := 1 TO iIloscDodanychPodzespolow DO
	IF (NOT arrOperacjaWykonana [i]) THEN
		arrOperacjaWykonana [i]				:= arrPodzesoly [i].SM_Resetting (eTrybPracy := eTrybPracy);
	END_IF
	bResetingOK								:= bResetingOK AND arrOperacjaWykonana [i];
END_FOR

IF (bResetingSkonczone OR bResetingOK) THEN
	eStan									:= E_PMLState.IDLE;
	bPierwszePrzejscieWOperacji				:= FALSE;
	bResetingSkonczone						:= FALSE;
	bResetingOK								:= FALSE;
ELSIF (bStop) THEN
	NacisnietyStopPrzejscieDoStopping ();
ELSIF (bAbort) THEN
	NacisnietyAbortPrzejscieDoAborting ();
END_IF
END_METHOD

//==================================================================================================
//								RJM Maszyny sp. z o.o.
//									13.05.2022
//	Obsługa stanu STARTING  
// 	v1.0	|| TC v 3.1.4024.29		|| - pierwsza wersja
//==================================================================================================
METHOD SM_Starting : BOOL
VAR_INPUT
END_VAR

VAR
	i										: INT;
	bStartingOK								: BOOL := TRUE;
END_VAR
IF (NOT bPierwszePrzejscieWOperacji) THEN
	FOR i := 1 TO iIloscDodanychPodzespolow DO
		arrOperacjaWykonana [i] 			:= FALSE;
	END_FOR
	bPierwszePrzejscieWOperacji				:= TRUE;
END_IF
FOR i := 1 TO iIloscDodanychPodzespolow DO
	IF (NOT arrOperacjaWykonana [i]) THEN
		arrOperacjaWykonana [i]				:= arrPodzesoly [i].SM_Starting ();
	END_IF
	bStartingOK								:= bStartingOK AND arrOperacjaWykonana [i];
END_FOR

IF (bStartingZakonczone OR bStartingOK) THEN
	bStartingZakonczone						:= FALSE;
	bPierwszePrzejscieWOperacji				:= FALSE;
	eStan									:= E_PMLState.EXECUTE;
ELSIF (bStop) THEN
	NacisnietyStopPrzejscieDoStopping ();
ELSIF (bAbort) THEN
	NacisnietyAbortPrzejscieDoAborting ();
END_IF
END_METHOD

//==================================================================================================
//								RJM Maszyny sp. z o.o.
//									13.05.2022
//	Obsługa stanu STOPPED  
// 	v1.0	|| TC v 3.1.4024.29		|| - pierwsza wersja
//==================================================================================================
METHOD SM_Stopped : BOOL
VAR_INPUT
END_VAR

VAR
	i: INT;
END_VAR
FOR i := 1 TO iIloscDodanychPodzespolow DO
	arrPodzesoly [i].SM_Stopped ();
END_FOR

IF (bReset) THEN
	eStan									:= E_PMLState.RESETTING;
END_IF
//ZMIANA TRYBU PRACY
IF (eTryb <> eTrybPracy) THEN
//	IF (iNumerTrybuPracy <>iPoprzedniTrybPracy) THEN
		eTrybPracy								:= eTryb;
		iPoprzedniTrybPracy						:= iNumerTrybuPracy;
		eStan									:= E_PMLState.ABORTING;
//	END_IF
END_IF
//ZMIANA TRYBU PRACY
END_METHOD

//==================================================================================================
//								RJM Maszyny sp. z o.o.
//									13.05.2022
//	Obsługa stanu STOPPING  
// 	v1.0	|| TC v 3.1.4024.29		|| - pierwsza wersja
//==================================================================================================
METHOD SM_Stopping : BOOL
VAR_INPUT
END_VAR

VAR
	i										: INT;
	bStoppingOK								: BOOL := TRUE;
END_VAR
IF (NOT bPierwszePrzejscieWOperacji) THEN
	FOR i := 1 TO iIloscDodanychPodzespolow DO
		arrOperacjaWykonana [i] 			:= FALSE;
	END_FOR
	bPierwszePrzejscieWOperacji				:= TRUE;
END_IF
FOR i := 1 TO iIloscDodanychPodzespolow DO
	IF (NOT arrOperacjaWykonana [i]) THEN
		arrOperacjaWykonana [i]				:= arrPodzesoly [i].SM_Stopping ();
	END_IF
	bStoppingOK								:= bStoppingOK AND arrOperacjaWykonana [i];
END_FOR

IF (bStoppingZakonczone OR bStoppingOK) THEN
	bStoppingZakonczone						:= FALSE;
	bPierwszePrzejscieWOperacji				:= FALSE;
	eStan									:= E_PMLState.STOPPED;
END_IF
END_METHOD

//==================================================================================================
//								RJM Maszyny sp. z o.o.
//									13.05.2022
//	Obsługa stanu SUSPENDED - praca wstrzymana prze operatora  
// 	v1.0	|| TC v 3.1.4024.29		|| - pierwsza wersja
//==================================================================================================
METHOD SM_Suspended : BOOL
VAR_INPUT
END_VAR
VAR
	i 										: INT;
END_VAR
FOR i := 1 TO iIloscDodanychPodzespolow DO
	arrPodzesoly [i].SM_Suspended ();
END_FOR

IF (bUnsuspend) THEN
	eStan									:= E_PMLState.UNSUSPENDING;
ELSIF (bStop) THEN
	NacisnietyStopPrzejscieDoStopping ();
ELSIF (bAbort) THEN
	NacisnietyAbortPrzejscieDoAborting ();
END_IF
END_METHOD

//==================================================================================================
//								RJM Maszyny sp. z o.o.
//									13.05.2022
//	Obsługa stanu SUSPENDING  
// 	v1.0	|| TC v 3.1.4024.29		|| - pierwsza wersja
//==================================================================================================
METHOD SM_Suspending : BOOL
VAR_INPUT
END_VAR

VAR
	i										: INT;
	bSuspendingOK							: BOOL := TRUE;
END_VAR
IF (NOT bPierwszePrzejscieWOperacji) THEN
	FOR i := 1 TO iIloscDodanychPodzespolow DO
		arrOperacjaWykonana [i] 			:= FALSE;
	END_FOR
	bPierwszePrzejscieWOperacji				:= TRUE;
END_IF
FOR i := 1 TO iIloscDodanychPodzespolow DO
	IF (NOT arrOperacjaWykonana [i]) THEN
		arrOperacjaWykonana [i]				:= arrPodzesoly [i].SM_Suspending ();
	END_IF
	bSuspendingOK							:= bSuspendingOK AND arrOperacjaWykonana [i];
END_FOR

IF (bSuspendingZakonczone OR bSuspendingOK) THEN
	bSuspendingZakonczone					:= FALSE;
	bPierwszePrzejscieWOperacji				:= FALSE;
	eStan									:= E_PMLState.SUSPENDED;
ELSIF (bStop) THEN
	NacisnietyStopPrzejscieDoStopping ();
ELSIF (bAbort) THEN
	NacisnietyAbortPrzejscieDoAborting ();
END_IF
END_METHOD

METHOD SM_Undefined : BOOL
VAR_INPUT
END_VAR
IF (bReset) THEN
	eStan									:= E_PMLState.ABORTING;
END_IF
END_METHOD

//==================================================================================================
//								RJM Maszyny sp. z o.o.
//									13.05.2022
//	Obsługa stanu UNHOLDING  
// 	v1.0	|| TC v 3.1.4024.29		|| - pierwsza wersja
//==================================================================================================
METHOD SM_Unholding : BOOL
VAR_INPUT
END_VAR

VAR
	i										: INT;
	bUnholdingOK							: BOOL := TRUE;
END_VAR
IF (NOT bPierwszePrzejscieWOperacji) THEN
	FOR i := 1 TO iIloscDodanychPodzespolow DO
		arrOperacjaWykonana [i] 			:= FALSE;
	END_FOR
	bPierwszePrzejscieWOperacji				:= TRUE;
END_IF
FOR i := 1 TO iIloscDodanychPodzespolow DO
	IF (NOT arrOperacjaWykonana [i]) THEN
		arrOperacjaWykonana [i]				:= arrPodzesoly [i].SM_Unholding ();
	END_IF
	bUnholdingOK							:= bUnholdingOK AND arrOperacjaWykonana [i];
END_FOR

IF (bUnholdingZakonczone OR bUnholdingOK) THEN
	bUnholdingZakonczone					:= FALSE;
	bPierwszePrzejscieWOperacji				:= FALSE;
	eStan									:= E_PMLState.EXECUTE;
ELSIF (bStop) THEN
	NacisnietyStopPrzejscieDoStopping ();
ELSIF (bAbort) THEN
	NacisnietyAbortPrzejscieDoAborting ();
END_IF
END_METHOD

//==================================================================================================
//								RJM Maszyny sp. z o.o.
//									13.05.2022
//	Obsługa stanu UNSUSPENDING  
// 	v1.0	|| TC v 3.1.4024.29		|| - pierwsza wersja
//==================================================================================================
METHOD SM_Unsuspending : BOOL
VAR_INPUT
END_VAR

VAR
	i										: INT;
	bUnsuspendingOK							: BOOL := TRUE;
END_VAR
IF (NOT bPierwszePrzejscieWOperacji) THEN
	FOR i := 1 TO iIloscDodanychPodzespolow DO
		arrOperacjaWykonana [i] 			:= FALSE;
	END_FOR
	bPierwszePrzejscieWOperacji				:= TRUE;
END_IF
FOR i := 1 TO iIloscDodanychPodzespolow DO
	IF (NOT arrOperacjaWykonana [i]) THEN
		arrOperacjaWykonana [i]				:= arrPodzesoly [i].SM_Unsuspending ();
	END_IF
	bUnsuspendingOK							:= bUnsuspendingOK AND arrOperacjaWykonana [i];
END_FOR

IF (bUnsuspendingZakonczone or bUnsuspendingOK) THEN
	bUnsuspendingZakonczone					:= FALSE;
	bPierwszePrzejscieWOperacji				:= FALSE;
	eStan									:= E_PMLState.EXECUTE;
ELSIF (bStop) THEN
	NacisnietyStopPrzejscieDoStopping ();
ELSIF (bAbort) THEN
	NacisnietyAbortPrzejscieDoAborting ();
END_IF
END_METHOD

//==================================================================================================
//								RJM Maszyny sp. z o.o.
//									13.05.2022
//	Stan pracy metoda sterująca  
// 	v1.0	|| TC v 3.1.4024.29		|| - pierwsza wersja
//==================================================================================================
METHOD PROTECTED StanMaszyny : BOOL
VAR_INPUT
END_VAR
iAktualnyStan 								:= eStan;
iNumerTrybuPracy							:= eTrybPracy;
IF (iAktualnyStan <> iPoprzedniStan) THEN
	arrVisuStany [iAktualnyStan].bAktywny 	:= TRUE;
	arrVisuStany [iPoprzedniStan].bAktywny	:= FALSE;
	iPoprzedniStan								:= iAktualnyStan;
END_IF


CASE eStan OF
	E_PMLState.UNDEFINED	:
		SM_Undefined ();
	E_PMLState.CLEARING 	:
		SM_Clearing ();
	E_PMLState.STOPPED 		:
		SM_Stopped ();
	E_PMLState.STARTING 	:
		SM_Starting ();
	E_PMLState.IDLE 		:
		SM_Idle ();
	E_PMLState.SUSPENDED 	:
		SM_Suspended ();
	E_PMLState.EXECUTE 		:
		SM_Execute (eTrybPracy := eTrybPracy);
	E_PMLState.STOPPING	 	:
		SM_Stopping ();
	E_PMLState.ABORTING 	:
		SM_Aborting ();
	E_PMLState.ABORTED 		:
		SM_Aborted ();
	E_PMLState.HOLDING 		:
		SM_Holding ();
	E_PMLState.HELD 		:
		SM_Held ();
	E_PMLState.UNHOLDING 	:
		SM_Unholding ();
	E_PMLState.SUSPENDING 	:
		SM_Suspending ();
	E_PMLState.UNSUSPENDING :
		SM_Unsuspending ();
	E_PMLState.RESETTING 	:
		SM_Resetting ();
	E_PMLState.COMPLETING 	:
		SM_Completing ();
	E_PMLState.COMPLETE	 	:
		SM_Complete ();
END_CASE
END_METHOD

//==================================================================================================
//								RJM Maszyny sp. z o.o.
//									13.05.2022
//	Zwraca stan pracy  
// 	v1.0	|| TC v 3.1.4024.29		|| - pierwsza wersja
//==================================================================================================
PROPERTY StanPracy : E_PMLState
GET
StanPracy									:= eStan;
END_GET
END_PROPERTY

//==================================================================================================
//								RJM Maszyny sp. z o.o.
//									13.05.2022
//	Zwraca tryb pracy  
// 	v1.0	|| TC v 3.1.4024.29		|| - pierwsza wersja
//==================================================================================================
PROPERTY TrybPracy : E_PMLUnitMode
GET
TrybPracy									:= eTrybPracy;
END_GET
END_PROPERTY

END_FUNCTION_BLOCK

// ---- POUs/91 - Elementy Sterujace/POU/FB_ElementySterujace.TcPOU
//==================================================================================================
//								RJM Maszyny sp. z o.o.
//									13.05.2022
//	Sterowanie elementami wizualnymi maszyny w zalezności od stanu pracy 
// 	v1.0	|| TC v 3.1.4024.29		|| - pierwsza wersja
//==================================================================================================
FUNCTION_BLOCK FB_ElementySterujace IMPLEMENTS ITF_StanMaszyny
VAR_INPUT

END_VAR
VAR_OUTPUT
END_VAR
VAR
	fbWieza									: ITF_WiezaSygnalizacyjna;
	fbPrzyciskStart							: ITF_Przycisk;
	fbPrzyciskStop							: ITF_Przycisk;
	eStanMaszyny							: E_PMLState;
	eStanMaszynyPoprzedni					: E_PMLState;
	eTrybPracy								: E_PMLUnitMode;
	
	fbImpulsyStart							: FB_Impulsy;
	tCzasZapaloneStart						: TIME;
	tCzasZgaszoneStart						: TIME;
	fbImpulsyStop							: FB_Impulsy;
	tCzasZapaloneStop						: TIME;
	tCzasZgaszoneStop						: TIME;
	
	bPodswietlanieStart						: BOOL;
	bPodswietlanieStop						: BOOL;
	bWlaczMiganieStart						: BOOL;
	bWlaczMiganieStop						: BOOL;
END_VAR

IF (eStanMaszyny <> eStanMaszynyPoprzedni) THEN
	CASE eStanMaszyny OF
		E_PMLState.UNDEFINED	:
	//		SM_Undefined ();
		E_PMLState.CLEARING 	:
			SM_Clearing ();
		E_PMLState.STOPPED 		:
			SM_Stopped ();
		E_PMLState.STARTING 	:
			SM_Starting ();
		E_PMLState.IDLE 		:
			SM_Idle ();
		E_PMLState.SUSPENDED 	:
			SM_Suspended ();
		E_PMLState.EXECUTE 		:
			SM_Execute (eTrybPracy := eTrybPracy);
		E_PMLState.STOPPING	 	:
			SM_Stopping ();
		E_PMLState.ABORTING 	:
			SM_Aborting ();
		E_PMLState.ABORTED 		:
			SM_Aborted ();
		E_PMLState.HOLDING 		:
			SM_Holding ();
		E_PMLState.HELD 		:
			SM_Held ();
		E_PMLState.UNHOLDING 	:
			SM_Unholding ();
		E_PMLState.SUSPENDING 	:
			SM_Suspending ();
		E_PMLState.UNSUSPENDING :
			SM_Unsuspending ();
		E_PMLState.RESETTING 	:
			SM_Resetting (eTrybPracy := eTrybPracy);
		E_PMLState.COMPLETING 	:
			SM_Completing ();
		E_PMLState.COMPLETE	 	:
			SM_Complete ();
	END_CASE
	eStanMaszynyPoprzedni						:= eStanMaszyny;
END_IF
fbImpulsyStart (bWlacz := bWlaczMiganieStart, tZapalone := tCzasZapaloneStart, tZgaszone := tCzasZgaszoneStart);
fbPrzyciskStart.Podswietlenie					:= bPodswietlanieStart AND 
													((bWlaczMiganieStart AND fbImpulsyStart.Wyjscie) OR NOT bWlaczMiganieStart);
fbImpulsyStop (bWlacz := bWlaczMiganieStop, tZapalone := tCzasZapaloneStop, tZgaszone := tCzasZgaszoneStop);
fbPrzyciskStop.Podswietlenie					:= bPodswietlanieStop AND 
													((bWlaczMiganieStop AND fbImpulsyStop.Wyjscie) OR NOT bWlaczMiganieStop);

METHOD FB_init : BOOL
VAR_INPUT
	bInitRetains : BOOL; // if TRUE, the retain variables are initialized (warm start / cold start)
	bInCopyCode : BOOL;  // if TRUE, the instance afterwards gets moved into the copy code (online change)
	fbWieza									: ITF_WiezaSygnalizacyjna;
	fbPrzyciskStart							: ITF_Przycisk;
	fbPrzyciskStop							: ITF_Przycisk;
END_VAR
THIS^.fbWieza								:= fbWieza;
THIS^.fbPrzyciskStart						:= fbPrzyciskStart;
THIS^.fbPrzyciskStop						:= fbPrzyciskStop;
END_METHOD

PROPERTY NacisnietyStart : BOOL
GET
NacisnietyStart								:= fbPrzyciskStart.CzyNacisniety;
END_GET
END_PROPERTY


PROPERTY NacisnietyStop : BOOL
GET
NacisnietyStop								:= fbPrzyciskStop.CzyNacisniety;
END_GET
END_PROPERTY

METHOD SM_Aborted : BOOL
VAR_INPUT

END_VAR
bWlaczMiganieStart							:= FALSE;
bPodswietlanieStart							:= FALSE;
bWlaczMiganieStop							:= FALSE;
bPodswietlanieStop							:= TRUE;
END_METHOD

METHOD SM_Aborting : BOOL
VAR_INPUT
END_VAR
tCzasZapaloneStart							:= T#500MS;
tCzasZgaszoneStart							:= T#500MS;
tCzasZapaloneStop							:= T#500MS;
tCzasZgaszoneStop							:= T#500MS;
	
bWlaczMiganieStart							:= TRUE;
bPodswietlanieStart							:= TRUE;
bWlaczMiganieStop							:= TRUE;
bPodswietlanieStop							:= TRUE;
END_METHOD

METHOD SM_Clearing : BOOL
VAR_INPUT
END_VAR
bWlaczMiganieStart							:= FALSE;
bPodswietlanieStart							:= FALSE;
bWlaczMiganieStop							:= FALSE;
bPodswietlanieStop							:= FALSE;
END_METHOD

METHOD SM_Complete : BOOL
VAR_INPUT
END_VAR

bWlaczMiganieStart							:= FALSE;
bPodswietlanieStart							:= FALSE;
bWlaczMiganieStop							:= FALSE;
bPodswietlanieStop							:= TRUE;
END_METHOD

METHOD SM_Completing : BOOL
VAR_INPUT
END_VAR
tCzasZapaloneStart							:= T#1000MS;
tCzasZgaszoneStart							:= T#500MS;
tCzasZapaloneStop							:= T#1000MS;
tCzasZgaszoneStop							:= T#500MS;
	
bWlaczMiganieStart							:= TRUE;
bPodswietlanieStart							:= TRUE;
bWlaczMiganieStop							:= FALSE;
bPodswietlanieStop							:= FALSE;
END_METHOD

METHOD SM_Execute : BOOL
VAR_INPUT
	eTrybPracy								: E_PMLUnitMode;
END_VAR
	
bWlaczMiganieStart							:= FALSE;
bPodswietlanieStart							:= TRUE;
bWlaczMiganieStop							:= FALSE;
bPodswietlanieStop							:= FALSE;
END_METHOD

METHOD SM_Held : BOOL
VAR_INPUT
END_VAR
tCzasZapaloneStart							:= T#1500MS;
tCzasZgaszoneStart							:= T#1000MS;
tCzasZapaloneStop							:= T#500MS;
tCzasZgaszoneStop							:= T#500MS;
	
bWlaczMiganieStart							:= TRUE;
bPodswietlanieStart							:= TRUE;
bWlaczMiganieStop							:= FALSE;
bPodswietlanieStop							:= FALSE;
END_METHOD

METHOD SM_Holding : BOOL
VAR_INPUT
END_VAR
tCzasZapaloneStart							:= T#1500MS;
tCzasZgaszoneStart							:= T#1000MS;
tCzasZapaloneStop							:= T#500MS;
tCzasZgaszoneStop							:= T#500MS;
	
bWlaczMiganieStart							:= TRUE;
bPodswietlanieStart							:= TRUE;
bWlaczMiganieStop							:= FALSE;
bPodswietlanieStop							:= FALSE;
END_METHOD

METHOD SM_Idle : BOOL
VAR_INPUT
END_VAR

	
bWlaczMiganieStart							:= FALSE;
bPodswietlanieStart							:= FALSE;
bWlaczMiganieStop							:= FALSE;
bPodswietlanieStop							:= TRUE;
END_METHOD

METHOD SM_Resetting : BOOL
VAR_INPUT
	eTrybPracy								: E_PMLUnitMode;
END_VAR

bWlaczMiganieStart							:= FALSE;
bPodswietlanieStart							:= FALSE;
bWlaczMiganieStop							:= FALSE;
bPodswietlanieStop							:= FALSE;
END_METHOD

METHOD SM_Starting : BOOL
VAR_INPUT
END_VAR
tCzasZapaloneStart							:= T#1500MS;
tCzasZgaszoneStart							:= T#1500MS;
tCzasZapaloneStop							:= T#500MS;
tCzasZgaszoneStop							:= T#500MS;
	
bWlaczMiganieStart							:= TRUE;
bPodswietlanieStart							:= TRUE;
bWlaczMiganieStop							:= FALSE;
bPodswietlanieStop							:= FALSE;
END_METHOD

METHOD SM_Stopped : BOOL
VAR_INPUT
END_VAR
tCzasZapaloneStart							:= T#1500MS;
tCzasZgaszoneStart							:= T#1000MS;
tCzasZapaloneStop							:= T#500MS;
tCzasZgaszoneStop							:= T#500MS;
	
bWlaczMiganieStart							:= FALSE;
bPodswietlanieStart							:= FALSE;
bWlaczMiganieStop							:= FALSE;
bPodswietlanieStop							:= TRUE;
END_METHOD

METHOD SM_Stopping : BOOL
VAR_INPUT
END_VAR
tCzasZapaloneStart							:= T#1500MS;
tCzasZgaszoneStart							:= T#1000MS;
tCzasZapaloneStop							:= T#1500MS;
tCzasZgaszoneStop							:= T#1000MS;
	
bWlaczMiganieStart							:= FALSE;
bPodswietlanieStart							:= FALSE;
bWlaczMiganieStop							:= TRUE;
bPodswietlanieStop							:= TRUE;
END_METHOD

METHOD SM_Suspended : BOOL
VAR_INPUT
END_VAR
tCzasZapaloneStart							:= T#2000MS;
tCzasZgaszoneStart							:= T#1500MS;
tCzasZapaloneStop							:= T#500MS;
tCzasZgaszoneStop							:= T#500MS;
	
bWlaczMiganieStart							:= TRUE;
bPodswietlanieStart							:= TRUE;
bWlaczMiganieStop							:= FALSE;
bPodswietlanieStop							:= FALSE;
END_METHOD

METHOD SM_Suspending : BOOL
VAR_INPUT
END_VAR
tCzasZapaloneStart							:= T#2000MS;
tCzasZgaszoneStart							:= T#1500MS;
tCzasZapaloneStop							:= T#500MS;
tCzasZgaszoneStop							:= T#500MS;
	
bWlaczMiganieStart							:= TRUE;
bPodswietlanieStart							:= TRUE;
bWlaczMiganieStop							:= FALSE;
bPodswietlanieStop							:= FALSE;
END_METHOD

METHOD SM_Unholding : BOOL
VAR_INPUT
END_VAR
tCzasZapaloneStart							:= T#1500MS;
tCzasZgaszoneStart							:= T#1000MS;
tCzasZapaloneStop							:= T#500MS;
tCzasZgaszoneStop							:= T#500MS;
	
bWlaczMiganieStart							:= TRUE;
bPodswietlanieStart							:= TRUE;
bWlaczMiganieStop							:= FALSE;
bPodswietlanieStop							:= FALSE;
END_METHOD

METHOD SM_Unsuspending : BOOL
VAR_INPUT
END_VAR
tCzasZapaloneStart							:= T#2000MS;
tCzasZgaszoneStart							:= T#1500MS;
tCzasZapaloneStop							:= T#500MS;
tCzasZgaszoneStop							:= T#500MS;
	
bWlaczMiganieStart							:= TRUE;
bPodswietlanieStart							:= TRUE;
bWlaczMiganieStop							:= FALSE;
bPodswietlanieStop							:= FALSE;
END_METHOD

PROPERTY StanMaszyny : E_PMLState
SET
eStanMaszyny								:= StanMaszyny;
END_SET
END_PROPERTY

PROPERTY TrybPracy : E_PMLUnitMode
SET
eTrybPracy									:= TrybPracy;
END_SET
END_PROPERTY

END_FUNCTION_BLOCK

// ---- POUs/92 - Elementy maszyny/Impulsy/POU/FB_Impulsy.TcPOU
FUNCTION_BLOCK FB_Impulsy
VAR_INPUT
	bWlacz									: BOOL;
	tZapalone								: TIME;
	tZgaszone								: TIME;
END_VAR
VAR_OUTPUT
END_VAR
VAR
	bWyjscie								: BOOL;
	tonZapalone								: TON;
	tonZgaszone								: TON;
END_VAR

IF (bWlacz) THEN
	tonZapalone (IN := NOT tonZgaszone.Q, PT := tZapalone);
	tonZgaszone (IN := tonZapalone.Q, PT := tZgaszone);
	
	IF (tonZapalone.Q) THEN
		bWyjscie								:= FALSE;
	ELSE
		bWyjscie								:= TRUE;
	END_IF
ELSE
	bWyjscie								:= FALSE;
END_IF

PROPERTY Wyjscie : BOOL
GET
Wyjscie									:= bWyjscie;
END_GET
END_PROPERTY

END_FUNCTION_BLOCK

// ---- POUs/95 - Logowanie bledow/POU/FB_LogowanieBledow.TcPOU
//==================================================================================================
//							RJM MASZYNY SP. Z O>O>
//									05.02.2022
//	Metoda sterujaca logowaniem bledow
// 	v1.0	|| TC v 3.1.4024.22		|| - pierwsza wersja
//==================================================================================================
FUNCTION_BLOCK FB_LogowanieBledow
VAR_INPUT
	arrZdarzeniaPamietane					: REFERENCE TO ARRAY [1..GVL_LogowanieBledow_Stale.MAX_ILOSC_ZDARZEN_ZAPAMIETANYCH] OF DUT_LogowanieBledow_Zapamietanych;
	iIloscZdarzenZapamietanych				: REFERENCE TO INT;
	bWyswietlanieTablicyAlarmow				: BOOL;
END_VAR
VAR_OUTPUT
END_VAR
VAR
	arrTablicaElementowWykonawczych 		: ARRAY [1..GVL_LogowanieBledow_Stale.MAX_ILOSC_ELEMENTOW] OF ITF_LogowanieBledow_ElementWykonawczy;
	iIloscDodanychElementow					: INT;	//ilość dodanych elementow wykonawczych, przypisać w deklaracji	
	iJezykID								: INT := 1045;	//id języka - domyślnie polski	

	iIloscDodanychWszystkichZdarzen 		: INT;			//ilosść dodanych zdarzeń globalnie
	
	bwypelnij								: BOOL;			//Wypełnienie tablic - wykonać na początku i po zmianie języka
	bDaneWypelnione							: BOOL := FALSE;//jak true mozna odczytywac stany podzespolow
	iI										: INT;
	iJ										: INT;
	
	arrTablicaDefinicjiZdarzen				: ARRAY [1..GVL_LogowanieBledow_Stale.MAX_ILOSC_ZDARZEN] OF DUT_LogowanieBledow_Zdarzenie;
	arrTablicaDefinicjiZdarzenOpis			: ARRAY [1..GVL_LogowanieBledow_Stale.MAX_ILOSC_ZDARZEN] OF DUT_LogowanieBledow_ZdarzenieOpis;
	arrTablicaDefinicjiZdarzenStan			: ARRAY [1..GVL_LogowanieBledow_Stale.MAX_ILOSC_ZDARZEN] OF DUT_LogowanieBledow_ZdarzenieStan;
	arrTablicaWyswietlana					: ARRAY [1..GVL_LOgowanieBledow_Stale.MAX_ILOSC_ZDARZEN_DO_WYSWIETLANIA] OF DUT_LogowanieBledow_ZdarzenieWyswietlane;
	arrPoczatekZdarzenia					: ARRAY [1..GVL_LogowanieBledow_Stale.MAX_ILOSC_ZDARZEN] OF R_TRIG;
	arrKoniecZdarzenia						: ARRAY [1..GVL_LogowanieBledow_Stale.MAX_ILOSC_ZDARZEN] OF F_TRIG;

	fbLocalSystemTime						: FB_LocalSystemTime;
	stAktualnyCzas							: TIMESTRUCT;				// Aktualny czas sytemowy w formie struktury
	dtAktualnyCzas							: DT;		
	bBladRozmiaruTablicyMozliwychZdarzen	: BOOL;						// Niewlasciwy rozmiar tablicy zdarzen - sprawdz HS_ILOSC_ZDARZEN_PAMIETANYCH
	bReferencjaOK							: BOOL;
	bInicjalizacjaDanychTablicyPamietanych	: BOOL := FALSE;
	tonOdswierzanieTablicyPamieci			: TON;
	tOdswierzenieTablicyPamieci				: TIME := T#100MS;
	bOdswierzanieCiagle						: BOOL;
	tonOdswierzaniaTablicyWyswietlania		: TON;
	tOdswierzaniaTablicyWyswietlania		: TIME := T#200MS;
	stWyswietlanieParametry					: DUT_LogowanieBledow_WyswietlanieParametry;
	bWiecejDanychZapamietanych				: BOOL;	//informacja ze jest wiecej danych zapamietanych niz do wyswietlenia
END_VAR

//Pobranie aktualnego czasu systemu
	fbLocalSystemTime (bEnable:= TRUE, systemTime=> stAktualnyCzas);
	dtAktualnyCzas								:= SYSTEMTIME_TO_DT(stAktualnyCzas);
//Sprawdzenie błędów rozmiaru tablic 
	bBladRozmiaruTablicyMozliwychZdarzen 		:= GVL_LogowanieBledow_Stale.MAX_ILOSC_ZDARZEN < 5 OR
													GVL_LogowanieBledow_Stale.MAX_ILOSC_ZDARZEN > 1000;
//Nie ma błędów pracuj z tablicami
	bReferencjaOK := __ISVALIDREF (arrZdarzeniaPamietane);

	IF (NOT bBladRozmiaruTablicyMozliwychZdarzen AND bReferencjaOK) THEN
	//Inicjalizacja tablicy przy starcie 
		Inicjalizacja ();
	//Wypełnienie tablicy zdarzen dla wszystkich elementow
		IF(bwypelnij) THEN
			WypelnianieTablicyZdarzen ();
		END_IF
	//Aktualizacja tablicy stanów
	//Timer odswiezania
		tonOdswierzanieTablicyPamieci(IN:= NOT tonOdswierzanieTablicyPamieci.Q, PT:= tOdswierzenieTablicyPamieci, Q=> , ET=> );
		IF (bDaneWypelnione AND (bOdswierzanieCiagle OR tonOdswierzanieTablicyPamieci.Q)) THEN
			ObslugaAktywnychZdarzen ();
		END_IF		
	//Odswierzanie tablicy alarmow
		tonOdswierzaniaTablicyWyswietlania(IN:= NOT tonOdswierzaniaTablicyWyswietlania.Q,
											 PT:= tOdswierzaniaTablicyWyswietlania, Q=> , ET=> );		// Timer odswiezania
		IF (bWyswietlanieTablicyAlarmow) THEN
			Wyswietlanie ();
		END_IF
	END_IF

METHOD FB_init : BOOL
VAR_INPUT
	bInitRetains : BOOL; // if TRUE, the retain variables are initialized (warm start / cold start)
	bInCopyCode : BOOL;  // if TRUE, the instance afterwards gets moved into the copy code (online change)
	tablica 								: ARRAY [1..GVL_LogowanieBledow_Stale.MAX_ILOSC_ELEMENTOW] OF ITF_LogowanieBledow_ElementWykonawczy;
	iIloscDodanychElementow					: INT;
END_VAR
THIS^.arrTablicaElementowWykonawczych 								:= tablica;
THIS^.iIloscDodanychElementow				:= iIloscDodanychElementow;
END_METHOD

//==================================================================================================
//							RJM MASZYNY SP. Z O>O>
//									05.02.2022
//	Inicjalizacja tablicy zapamietanych zdarzen
//	Wyszukanie niezakonczonych i konczymy
// 	v1.0	|| TC v 3.1.4024.22		|| - pierwsza wersja
//==================================================================================================
METHOD PRIVATE Inicjalizacja : BOOL
VAR_INPUT
END_VAR
		IF (NOT bInicjalizacjaDanychTablicyPamietanych) THEN
			bInicjalizacjaDanychTablicyPamietanych	:= TRUE;
			FOR iJ := 1 TO iIloscZdarzenZapamietanych DO
				IF (arrZdarzeniaPamietane [iJ].bAktywne) THEN
					arrZdarzeniaPamietane [iJ].bAktywne	:= FALSE;
					//wywolac ZadanieKonie();
				END_IF
			END_FOR
		END_IF
END_METHOD

//==================================================================================================
//							RJM MASZYNY SP. Z O>O>
//									05.02.2022
//	Skanowanie tablicy stanow i po pojawieniu sie aktywnego zdarzenia dodajemy do tablicy pamietanych
//	po zakonczeniu aktywnosci zgloszenia zmieniamy w tablicy pamietanych
// 	v1.0	|| TC v 3.1.4024.22		|| - pierwsza wersja
//==================================================================================================
METHOD PRIVATE ObslugaAktywnychZdarzen : BOOL
VAR_INPUT
END_VAR
	FOR iJ := 1 TO iIloscDodanychElementow DO
		arrTablicaElementowWykonawczych [iJ].ZwrocTabliceStanu (arrTablicaDefinicjiZdarzenStan := arrTablicaDefinicjiZdarzenStan);
	END_FOR
	
	FOR iJ := 1 TO iIloscDodanychWszystkichZdarzen DO
		arrPoczatekZdarzenia [iJ] (CLK := arrTablicaDefinicjiZdarzenStan [iJ].bAktywne);
		IF (arrPoczatekZdarzenia [iJ].Q) THEN
		//dodac nowe zdarzenie do tablicy arrZdarzeniaPamietane
			ZdarzeniePoczatek (iIdZdarzenia 	:= arrTablicaDefinicjiZdarzen [iJ].iIdZdarzenia,
								dtAktualnyCzas 	:= dtAktualnyCzas);
		END_IF
		arrKoniecZdarzenia [iJ] (CLK := arrTablicaDefinicjiZdarzenStan [iJ].bAktywne);
		IF (arrKoniecZdarzenia [iJ].Q) THEN
		//odznaczyc koniec zdarzenia w tablicy arrZdarzeniaPamietane
			ZdarzenieKoniec (iNumerWiersza 		:= ZnajdzZdarzenieWTablicyPamietanychPoID (iIDZdarzenia := arrTablicaDefinicjiZdarzen [iJ].iIdZdarzenia),
								dtAktualnyCzas 	:= dtAktualnyCzas);
		END_IF
	END_FOR
END_METHOD

//==================================================================================================
//							RJM MASZYNY SP. Z O>O>
//									05.02.2022
//	Pobieranie danych zdarzen od podelementow systemu i dopisywanie ich do tablicy zdarzen
// 	v1.0	|| TC v 3.1.4024.22		|| - pierwsza wersja
//==================================================================================================
METHOD PRIVATE WypelnianieTablicyZdarzen : BOOL
VAR_INPUT
END_VAR
	bDaneWypelnione						:= FALSE;
	FOR iI := 1 TO iIloscDodanychElementow DO 
		arrTablicaElementowWykonawczych [iI].ZwrocTabliceDefinicji (	
												arrTablicaDefinicjiZdarzen := arrTablicaDefinicjiZdarzen,
												arrTablicaDefinicjiZdarzenOpis := arrTablicaDefinicjiZdarzenOpis,
												arrTablicaDefinicjiZdarzenStan := arrTablicaDefinicjiZdarzenStan,
												iIdZdarzenia := iIloscDodanychWszystkichZdarzen, 
												iNrPodzespolu := iI, 
												iNrPodelementu := 1,
												iNrElementu := 1, 
												iJezykId := iJezykID);
	END_FOR
	bwypelnij 							:= FALSE;
	bDaneWypelnione						:= TRUE;
END_METHOD

//==================================================================================================
//							RJM MASZYNY SP. Z O>O>
//									05.02.2022
//	Start wypelniania tablicy zdarzen
// 	v1.0	|| TC v 3.1.4024.22		|| - pierwsza wersja
//==================================================================================================
PROPERTY WypelnijTabliceZdarzen : BOOL
SET
bwypelnij									:= WypelnijTabliceZdarzen;
END_SET
END_PROPERTY

METHOD PRIVATE Wyswietlanie : BOOL
VAR_INPUT
END_VAR

VAR
	j										: INT;
	i										: INT;
	bUsunZWyswietlania						: BOOL;
END_VAR
IF (tonOdswierzaniaTablicyWyswietlania.Q) THEN
	MEMSET(ADR(arrTablicaWyswietlana),0,SIZEOF(arrTablicaWyswietlana));
	j										:= 1; //wskaznik wierszy tablicy wyswietlania
	bWiecejDanychZapamietanych				:= FALSE;
	FOR i := 1 TO iIloscZdarzenZapamietanych DO
		bUsunZWyswietlania					:= FALSE;	
		IF (arrZdarzeniaPamietane [i].iIDZdarzenia <> 0) THEN	//sprawdzenie czy w wierszu sa jakies dane
			//Ustawienie filtrow wyswietlania
			bUsunZWyswietlania				:= stWyswietlanieParametry.bFiltrID AND stWyswietlanieParametry.iFiltrID <> arrTablicaDefinicjiZdarzen [arrZdarzeniaPamietane [i].iIDZdarzenia].byRodzajZdarzenia;
//			bUsunZWyswietlania				:= bUsunZWyswietlania OR (stWyswietlanieParametry.bFiltrRodzaj AND stWyswietlanieParametry.byFiltrRodzaj <> arrTablicaDefinicjiZdarzen [arrZdarzeniaPamietane [i].iIDZdarzenia].byRodzajZdarzenia);
			bUsunZWyswietlania				:= bUsunZWyswietlania OR (stWyswietlanieParametry.bFiltrStartOD AND arrZdarzeniaPamietane [i].dtDataStart <= stWyswietlanieParametry.dtFiltrStartOD);
			bUsunZWyswietlania				:= bUsunZWyswietlania OR (stWyswietlanieParametry.bFiltrStartDO AND arrZdarzeniaPamietane [i].dtDataStart >= stWyswietlanieParametry.dtFiltrStartDO);
			bUsunZWyswietlania				:= bUsunZWyswietlania OR (stWyswietlanieParametry.bFiltrKoniecOD AND arrZdarzeniaPamietane [i].dtDataKoniec <= stWyswietlanieParametry.dtFiltrKoniecOD);
			bUsunZWyswietlania				:= bUsunZWyswietlania OR (stWyswietlanieParametry.bFiltrKoniecDO AND arrZdarzeniaPamietane [i].dtDataKoniec >= stWyswietlanieParametry.dtFiltrKoniecDO);
			bUsunZWyswietlania				:= bUsunZWyswietlania OR (stWyswietlanieParametry.bFiltrAktywne AND DT#1970-1-1-0:0:0 <> arrZdarzeniaPamietane[i].dtDataKoniec);
			// Analogicznie dodajemy inne filtry jesli jest taka potrzeba
			// Jesli element nie zostal usuniety przez filtr to dodajemy go do tablicy alarmow wyswietlanych
			IF (NOT bUsunZWyswietlania) THEN
				arrTablicaWyswietlana [j].sNrKomponentu	:= arrTablicaDefinicjiZdarzen [i].sNrKomponentu;
				arrTablicaWyswietlana [j].byRodzajZdarzenia	:= arrTablicaDefinicjiZdarzen [i].byRodzajZdarzenia;
 				arrTablicaWyswietlana [j].sOpis			:= arrTablicaDefinicjiZdarzenOpis [i].sOpis;
				arrTablicaWyswietlana [j].sKodBledu		:= arrTablicaDefinicjiZdarzen [i].sKodBledu;
				arrTablicaWyswietlana [j].dtDataStart	:= arrZdarzeniaPamietane [i].dtDataStart;
				arrTablicaWyswietlana [j].dtDataKoniec	:= arrZdarzeniaPamietane [i].dtDataKoniec;
				CASE arrTablicaWyswietlana [j].byRodzajZdarzenia OF
					1	: arrTablicaWyswietlana [j].dwKolor	:= 16#FFFF0000;	// blad 		- czerwony
					2	: arrTablicaWyswietlana [j].dwKolor	:= 16#FFFFFF00;	// ostzrezenie 	- zolty
					3	: arrTablicaWyswietlana [j].dwKolor	:= 16#FFFFFFFF;	// wiadomosc 	- bialy
					4	: arrTablicaWyswietlana [j].dwKolor	:= 16#FF0000FF; // safety 		- niebieski
				END_CASE
				j := j + 1;
			END_IF
		END_IF
		IF (j > GVL_LogowanieBledow_Stale.MAX_ILOSC_ZDARZEN_DO_WYSWIETLANIA) THEN
			bWiecejDanychZapamietanych		:= TRUE;
			EXIT;
		END_IF
	END_FOR
END_IF
END_METHOD

//==================================================================================================
//							RJM MASZYNY SP. Z O>O>
//									05.02.2022
//	Zdarzenie przestalo byc aktywne zmien dane
// 	v1.0	|| TC v 3.1.4024.22		|| - pierwsza wersja
//==================================================================================================
METHOD PRIVATE ZdarzenieKoniec : BOOL
VAR_INPUT
	iNumerWiersza							: INT;	//numer wiersza dla konkretnego IDzdarzenia
	dtAktualnyCzas							: DT;
END_VAR
arrZdarzeniaPamietane [iNumerWiersza].dtDataKoniec	:= dtAktualnyCzas;
arrZdarzeniaPamietane [iNumerWiersza].bAktywne		:= FALSE;
END_METHOD

//==================================================================================================
//							RJM MASZYNY SP. Z O>O>
//									05.02.2022
//	Dodanie nowego aktywnego zdarzenia do tablicy pamietanych
// 	v1.0	|| TC v 3.1.4024.22		|| - pierwsza wersja
//==================================================================================================
METHOD PRIVATE ZdarzeniePoczatek : BOOL
VAR_INPUT
	iIdZdarzenia							: INT;
	dtAktualnyCzas							: DT;
END_VAR
VAR
	i										: INT;
END_VAR
iIloscZdarzenZapamietanych					:= iIloscZdarzenZapamietanych + 1;
// Przesun elemety tablicy
FOR i := 0 TO iIloscZdarzenZapamietanych - 2 DO
	arrZdarzeniaPamietane [iIloscZdarzenZapamietanych - i]	:= arrZdarzeniaPamietane [iIloscZdarzenZapamietanych - i - 1];
END_FOR

// Dodaj nowy
//arrZdarzeniaPamietane [1].dwIDZdarzenia		:= stZdarzenie.dwIDZdarzenia;
arrZdarzeniaPamietane [1].iIDZdarzenia		:= iIDZdarzenia;
arrZdarzeniaPamietane [1].dtDataStart		:= dtAktualnyCzas;
arrZdarzeniaPamietane [1].dtDataKoniec		:= DT#1970-1-1-0:0:0;
arrZdarzeniaPamietane [1].bAktywne			:= TRUE;
END_METHOD

//==================================================================================================
//							RJM MASZYNY SP. Z O>O>
//									05.02.2022
//	Zwraca numer wiersza w tabeli pamieci z podanym idzdarzenia
// 	v1.0	|| TC v 3.1.4024.22		|| - pierwsza wersja
//==================================================================================================

METHOD PROTECTED ZnajdzZdarzenieWTablicyPamietanychPoID : INT
VAR_INPUT
	iIDZdarzenia							: INT;
END_VAR
VAR 
	i										: INT;
END_VAR
FOR i := 1 TO iIloscZdarzenZapamietanych DO
	IF (arrZdarzeniaPamietane [i].iIDZdarzenia = iIDZdarzenia) THEN
		ZnajdzZdarzenieWTablicyPamietanychPoID	:= i;
		EXIT;
	END_IF
END_FOR
END_METHOD

END_FUNCTION_BLOCK

// ---- POUs/01 - Elementy/Czujnik/POU/FB_Czujnik_NC.TcPOU
//==================================================================================================
//								RJM Maszyny sp. z o.o.
//									04.06.2022
//	Obsługa czujnika NC
// 	v1.0	|| TC v 3.1.4024.22		|| - pierwsza wersja
//==================================================================================================
FUNCTION_BLOCK FB_Czujnik_NC IMPLEMENTS ITF_Czujnik
VAR_INPUT
	bSymulacja								: BOOL;
END_VAR
VAR
	bWejscie						AT %I*	: BOOL;
END_VAR

//==================================================================================================
//								RJM Maszyny sp. z o.o.
//									04.06.2022
//	Obsługa czujnika  
// 	v1.0	|| TC v 3.1.4024.22		|| - pierwsza wersja
//==================================================================================================
PROPERTY CzyZadzialany : BOOL
GET
CzyZadzialany								:= NOT bWejscie;
END_GET
END_PROPERTY

END_FUNCTION_BLOCK

// ---- POUs/01 - Elementy/Elektrozawór/POU/FB_Elektrozawor_5na2_1Cewka.TcPOU
//==================================================================================================
//								RJM Maszyny sp. z o.o.
//									04.06.2022
//	Sterowanie elektrozaworem  - 5 na 2 z jedną cewką
// 	v1.0	|| TC v 3.1.4024.22		|| - pierwsza wersja
//==================================================================================================
FUNCTION_BLOCK FB_Elektrozawor_5na2_1Cewka IMPLEMENTS ITF_Elektozawor
VAR
	bCewkaA							AT %Q*	: BOOL;		//Cewka sterująca wyjściem 2 - do MAX
END_VAR

(*==================================================================================================
								RJM Maszyny sp. z o.o.
									04.06.2022
	Sterowanie cewkami elektrozaworu 
 	v1.0	|| TC v 3.1.4024.22		|| - pierwsza wersja
==================================================================================================*)
METHOD Steruj : BOOL
VAR_INPUT
	bKierunekWstrone0						: BOOL;
	bKierunekWStroneMax						: BOOL;
END_VAR
IF (bKierunekWStroneMax AND NOT bCewkaA) THEN
	bCewkaA									:= TRUE;
END_IF
IF  (bKierunekWstrone0 AND bCewkaA) THEN
	bCewkaA									:= FALSE;
END_IF
END_METHOD

END_FUNCTION_BLOCK

// ---- POUs/01 - Elementy/Elektrozawór/POU/FB_Elektrozawor_5na3_Odpowietrzony.TcPOU
//==================================================================================================
//								RJM Maszyny sp. z o.o.
//									04.06.2022
//	Sterowanie elektrozaworem  - 5 na 3 odpowietrzony 
//	nie mapodanych sygnałów na cewki powietrze nie jest podawane na siłownik
// 	v1.0	|| TC v 3.1.4024.22		|| - pierwsza wersja
//==================================================================================================
FUNCTION_BLOCK FB_Elektrozawor_5na3_Odpowietrzony IMPLEMENTS ITF_Elektozawor
VAR
	bCewkaA							AT %Q*	: BOOL;		//Cewka sterująca wyjściem 2 - 0 do MAX
	bCewkaB							AT %Q*	: BOOL;		//Cewka sterująca wyjściem 4 - MAX do 0
END_VAR

(*==================================================================================================
								RJM Maszyny sp. z o.o.
									04.06.2022
	Sterowanie cewkami elektrozaworu 
 	v1.0	|| TC v 3.1.4024.22		|| - pierwsza wersja
==================================================================================================*)
METHOD Steruj : BOOL
VAR_INPUT
	bKierunekWstrone0						: BOOL;
	bKierunekWStroneMax						: BOOL;
END_VAR
IF (bKierunekWStroneMax AND NOT bCewkaA) THEN
	bCewkaA									:= TRUE;
END_IF
IF  (bKierunekWstrone0 AND bCewkaA) THEN
	bCewkaA									:= FALSE;
END_IF

IF (bKierunekWstrone0 AND NOT bCewkaB) THEN
	bCewkaB									:= TRUE;
END_IF
IF  (bKierunekWStroneMax AND bCewkaB) THEN
	bCewkaB									:= FALSE;
END_IF
END_METHOD

END_FUNCTION_BLOCK

// ---- POUs/01 - Elementy/Elektrozawór/POU/FB_Elektrozawor_5na3_Zapowietrzony.TcPOU
//==================================================================================================
//								RJM Maszyny sp. z o.o.
//									04.06.2022
//	Sterowanie elektrozaworem  - 5 na 3 zapowietrzony 
//	nie ma podanych sygnałów na cewki powietrze jest podawane na siłownik (sterowanie odwrotne)
// 	v1.0	|| TC v 3.1.4024.22		|| - pierwsza wersja
//==================================================================================================
FUNCTION_BLOCK FB_Elektrozawor_5na3_Zapowietrzony IMPLEMENTS ITF_Elektozawor
VAR
	bCewkaA							AT %Q*	: BOOL;		//Cewka sterująca wyjściem 2 - 0 do MAX
	bCewkaB							AT %Q*	: BOOL;		//Cewka sterująca wyjściem 4 - MAX do 0
END_VAR

(*==================================================================================================
								RJM Maszyny sp. z o.o.
									04.06.2022
	Sterowanie cewkami elektrozaworu 
 	v1.0	|| TC v 3.1.4024.22		|| - pierwsza wersja
==================================================================================================*)
METHOD Steruj : BOOL
VAR_INPUT
	bKierunekWstrone0						: BOOL;
	bKierunekWStroneMax						: BOOL;
END_VAR
IF (bKierunekWStroneMax AND NOT bCewkaA) THEN
	bCewkaB									:= TRUE;
END_IF
IF  (bKierunekWstrone0 AND bCewkaA) THEN
	bCewkaB									:= FALSE;
END_IF

IF (bKierunekWstrone0 AND NOT bCewkaB) THEN
	bCewkaA									:= TRUE;
END_IF
IF  (bKierunekWStroneMax AND bCewkaB) THEN
	bCewkaA									:= FALSE;
END_IF
END_METHOD

END_FUNCTION_BLOCK

// ---- POUs/50 - testowy podzespol/POU/FB_TestowyPodzespol.TcPOU
FUNCTION_BLOCK FB_TestowyPodzespol IMPLEMENTS ITF_StanMaszyny
VAR_INPUT
END_VAR
VAR_OUTPUT
END_VAR
VAR
	bTest: BOOL;
END_VAR

METHOD SM_Aborted : BOOL
END_METHOD

METHOD SM_Aborting : BOOL
END_METHOD

METHOD SM_Clearing : BOOL
END_METHOD

METHOD SM_Complete : BOOL
END_METHOD

METHOD SM_Completing : BOOL
END_METHOD

METHOD SM_Execute : BOOL
END_METHOD

METHOD SM_Held : BOOL
END_METHOD

METHOD SM_Holding : BOOL
END_METHOD

METHOD SM_Idle : BOOL
END_METHOD


METHOD SM_Resetting : BOOL
IF (bTest) THEN
	SM_Resetting							:= TRUE;
ELSE
	SM_Resetting							:= FALSE;
END_IF
END_METHOD

METHOD SM_Starting : BOOL
END_METHOD

METHOD SM_Stopped : BOOL
END_METHOD

METHOD SM_Stopping : BOOL
END_METHOD

METHOD SM_Suspended : BOOL
END_METHOD

METHOD SM_Suspending : BOOL
END_METHOD

METHOD SM_Unholding : BOOL
END_METHOD

METHOD SM_Unsuspending : BOOL
END_METHOD

END_FUNCTION_BLOCK

// ---- POUs/51 - Krajalnica/POU/FB_Krajalnica_Komunikacja.TcPOU
FUNCTION_BLOCK FB_Krajalnica_Komunikacja EXTENDS FB_LogowanieBledow_ElementZlozony
VAR_INPUT
END_VAR
VAR_OUTPUT
END_VAR
VAR
END_VAR

METHOD DefinicjaTabeliZdarzen_1031_Niemiecki : BOOL
VAR_INPUT
	arrTablicaDefinicjiZdarzenOpis			: REFERENCE TO ARRAY [1..GVL_LogowanieBledow_Stale.MAX_ILOSC_ZDARZEN] OF DUT_LogowanieBledow_ZdarzenieOpis;

END_VAR
//arrTablicaDefinicjiZdarzenOpis [iStartId+0].sOpis	:= 'DE - TESTOWA WIADOMOSC';
END_METHOD

METHOD DefinicjaTabeliZdarzen_1033_Angielski : BOOL
VAR_INPUT
	arrTablicaDefinicjiZdarzenOpis			: REFERENCE TO ARRAY [1..GVL_LogowanieBledow_Stale.MAX_ILOSC_ZDARZEN] OF DUT_LogowanieBledow_ZdarzenieOpis;

END_VAR
//arrTablicaDefinicjiZdarzenOpis [iStartId+0].sOpis	:= 'EN - TESTOWA WIADOMOSC';
END_METHOD

METHOD DefinicjaTabeliZdarzen_1045_Polski : BOOL
VAR_INPUT
	arrTablicaDefinicjiZdarzenOpis			: REFERENCE TO ARRAY [1..GVL_LogowanieBledow_Stale.MAX_ILOSC_ZDARZEN] OF DUT_LogowanieBledow_ZdarzenieOpis;

END_VAR
//arrTablicaDefinicjiZdarzenOpis [iStartId+0].sOpis	:= 'PL - TESTOWA WIADOMOSC';
END_METHOD

METHOD DefinicjaTabeliZdarzen_Ogolna : BOOL
VAR_INPUT
	arrTablicaDefinicjiZdarzen				: REFERENCE TO ARRAY [1..GVL_LogowanieBledow_Stale.MAX_ILOSC_ZDARZEN] OF DUT_LogowanieBledow_Zdarzenie;
	arrTablicaDefinicjiZdarzenOpis			: REFERENCE TO ARRAY [1..GVL_LogowanieBledow_Stale.MAX_ILOSC_ZDARZEN] OF DUT_LogowanieBledow_ZdarzenieOpis;
	arrTablicaDefinicjiZdarzenStan			: REFERENCE TO ARRAY [1..GVL_LogowanieBledow_Stale.MAX_ILOSC_ZDARZEN] OF DUT_LogowanieBledow_ZdarzenieStan;

	iIdZdarzenia							: REFERENCE TO INT;
	iNrPodzespolu							: INT := 0;
	iNrPodelementu							: INT := 0;
	iNrElementu								: INT := 0;
END_VAR
(*
//testowy blad
	iIdZdarzenia												:= iIdZdarzenia + 1;
	arrTablicaDefinicjiZdarzen [iIdZdarzenia].iIdZdarzenia		:= iIdZdarzenia;
	arrTablicaDefinicjiZdarzen [iIdZdarzenia].byRodzajZdarzenia	:= 3;
	arrTablicaDefinicjiZdarzen [iIdZdarzenia].sKodBledu			:= '0001';
	arrTablicaDefinicjiZdarzen [iIdZdarzenia].sNrKomponentu		:= GenerujNrKomponentu (iNrPodzespolu := iNrPodzespolu, iNrPodelementu := iNrPodelementu, iNrElementu := iNrElementu); 
	arrTablicaDefinicjiZdarzenOpis [iIdZdarzenia].iIdZdarzenia 	:= iIdZdarzenia;
	arrTablicaDefinicjiZdarzenStan [iIdZdarzenia].iIdZdarzenia 	:= iIdZdarzenia;
	arrTablicaDefinicjiZdarzenStan [iIdZdarzenia].bAktywne		:= FALSE;
	*)
END_METHOD

END_FUNCTION_BLOCK

// ---- POUs/90 - Stan Maszyny/POU/FB_StanMaszyny_Baza.TcPOU
//==================================================================================================
//								RJM Maszyny sp. z o.o.
//									13.05.2022
//	Klasa bazowa dla podzespołów maszyny 
// 	v1.0	|| TC v 3.1.4024.29		|| - pierwsza wersja
//==================================================================================================
FUNCTION_BLOCK FB_StanMaszyny_Baza IMPLEMENTS ITF_StanMaszyny
VAR_INPUT
END_VAR
VAR_OUTPUT
END_VAR
VAR

END_VAR

//==================================================================================================
//								RJM Maszyny sp. z o.o.
//									13.05.2022
//	Obsługa stanu ABORTED  
// 	v1.0	|| TC v 3.1.4024.29		|| - pierwsza wersja
//==================================================================================================
METHOD SM_Aborted : BOOL
VAR_INPUT
END_VAR
END_METHOD

//==================================================================================================
//								RJM Maszyny sp. z o.o.
//									13.05.2022
//	Obsługa stanu ABORTING
// 	v1.0	|| TC v 3.1.4024.29		|| - pierwsza wersja
//==================================================================================================
METHOD SM_Aborting : BOOL
VAR_INPUT
END_VAR
END_METHOD

//==================================================================================================
//								RJM Maszyny sp. z o.o.
//									13.05.2022
//	Obsługa stanu CLEARING  
// 	v1.0	|| TC v 3.1.4024.29		|| - pierwsza wersja
//==================================================================================================
METHOD SM_Clearing : BOOL
VAR_INPUT
END_VAR
END_METHOD

//==================================================================================================
//								RJM Maszyny sp. z o.o.
//									13.05.2022
//	Obsługa stanu COMPLETE  
// 	v1.0	|| TC v 3.1.4024.29		|| - pierwsza wersja
//==================================================================================================
METHOD SM_Complete : BOOL
VAR_INPUT
END_VAR
END_METHOD

//==================================================================================================
//								RJM Maszyny sp. z o.o.
//									13.05.2022
//	Obsługa stanu COMPLITING  
// 	v1.0	|| TC v 3.1.4024.29		|| - pierwsza wersja
//==================================================================================================
METHOD SM_Completing : BOOL
VAR_INPUT
END_VAR
END_METHOD

//==================================================================================================
//								RJM Maszyny sp. z o.o.
//									13.05.2022
//	Obsługa stanu EXECUTE  
// 	v1.0	|| TC v 3.1.4024.29		|| - pierwsza wersja
//==================================================================================================
METHOD SM_Execute : BOOL
VAR_INPUT
END_VAR
END_METHOD

//==================================================================================================
//								RJM Maszyny sp. z o.o.
//									13.05.2022
//	Obsługa stanu HELD  
// 	v1.0	|| TC v 3.1.4024.29		|| - pierwsza wersja
//==================================================================================================
METHOD SM_Held : BOOL
VAR_INPUT
END_VAR
END_METHOD

//==================================================================================================
//								RJM Maszyny sp. z o.o.
//									13.05.2022
//	Obsługa stanu HOLDING - wsztrymanie pracy przez maszyne  
// 	v1.0	|| TC v 3.1.4024.29		|| - pierwsza wersja
//==================================================================================================
METHOD SM_Holding : BOOL
VAR_INPUT
END_VAR
END_METHOD

//==================================================================================================
//								RJM Maszyny sp. z o.o.
//									13.05.2022
//	Obsługa stanu IDLE - maszyna gotowado pracy  
// 	v1.0	|| TC v 3.1.4024.29		|| - pierwsza wersja
//==================================================================================================
METHOD SM_Idle : BOOL
VAR_INPUT
END_VAR
END_METHOD

//==================================================================================================
//								RJM Maszyny sp. z o.o.
//									13.05.2022
//	Obsługa stanu RESETTING  
// 	v1.0	|| TC v 3.1.4024.29		|| - pierwsza wersja
//==================================================================================================
METHOD SM_Resetting : BOOL
VAR_INPUT
END_VAR
END_METHOD

//==================================================================================================
//								RJM Maszyny sp. z o.o.
//									13.05.2022
//	Obsługa stanu STARTING  
// 	v1.0	|| TC v 3.1.4024.29		|| - pierwsza wersja
//==================================================================================================
METHOD SM_Starting : BOOL
VAR_INPUT
END_VAR
END_METHOD

//==================================================================================================
//								RJM Maszyny sp. z o.o.
//									13.05.2022
//	Obsługa stanu STOPPED  
// 	v1.0	|| TC v 3.1.4024.29		|| - pierwsza wersja
//==================================================================================================
METHOD SM_Stopped : BOOL
VAR_INPUT
END_VAR
END_METHOD

//==================================================================================================
//								RJM Maszyny sp. z o.o.
//									13.05.2022
//	Obsługa stanu STOPPING  
// 	v1.0	|| TC v 3.1.4024.29		|| - pierwsza wersja
//==================================================================================================
METHOD SM_Stopping : BOOL
VAR_INPUT
END_VAR
END_METHOD

//==================================================================================================
//								RJM Maszyny sp. z o.o.
//									13.05.2022
//	Obsługa stanu SUSPENDED - praca wstrzymana prze operatora  
// 	v1.0	|| TC v 3.1.4024.29		|| - pierwsza wersja
//==================================================================================================
METHOD SM_Suspended : BOOL
VAR_INPUT
END_VAR
END_METHOD

//==================================================================================================
//								RJM Maszyny sp. z o.o.
//									13.05.2022
//	Obsługa stanu SUSPENDING  
// 	v1.0	|| TC v 3.1.4024.29		|| - pierwsza wersja
//==================================================================================================
METHOD SM_Suspending : BOOL
VAR_INPUT
END_VAR
END_METHOD

//==================================================================================================
//								RJM Maszyny sp. z o.o.
//									13.05.2022
//	Obsługa stanu UNHOLDING  
// 	v1.0	|| TC v 3.1.4024.29		|| - pierwsza wersja
//==================================================================================================
METHOD SM_Unholding : BOOL
VAR_INPUT
END_VAR
END_METHOD

//==================================================================================================
//								RJM Maszyny sp. z o.o.
//									13.05.2022
//	Obsługa stanu UNSUSPENDING  
// 	v1.0	|| TC v 3.1.4024.29		|| - pierwsza wersja
//==================================================================================================
METHOD SM_Unsuspending : BOOL
VAR_INPUT
END_VAR
END_METHOD

END_FUNCTION_BLOCK

// ---- POUs/92 - Elementy maszyny/Przycisk/POU/FB_Przycisk_NC.TcPOU
//==================================================================================================
//								RJM Maszyny sp. z o.o.
//									22.06.2022
//	Obsługa przycisku ze stykiem NC
// 	v1.0	|| TC v 3.1.4024.22		|| - pierwsza wersja
//==================================================================================================
FUNCTION_BLOCK FB_Przycisk_NC IMPLEMENTS ITF_Przycisk
VAR
	bStyk							AT %I*	: BOOL;
	bPodswietlenie					AT %Q*	: BOOL;
END_VAR

PROPERTY CzyNacisniety : BOOL
GET
CzyNacisniety								:= NOT bStyk;
END_GET
END_PROPERTY

PROPERTY Podswietlenie : BOOL
SET
bPodswietlenie								:= Podswietlenie;
END_SET
END_PROPERTY

END_FUNCTION_BLOCK

// ---- GlobalTextList.TcGTLO
TEXTLIST GlobalTextList
  900 = '%s'
  977 = 'Abort'
  993 = 'Admin'
  970 = 'Bazuj ciecie 1'
  30 = 'Bazuj ciecie 2'
  176 = 'Bazuj Podawanie'
  836 = 'Bezpieczeństwo'
  340 = 'Błędy'
  322 = 'C1'
  888 = 'C1- bazowanie'
  11 = 'C1- ciecie'
  750 = 'C1- podawanie'
  655 = 'C2'
  746 = 'C2- bazowanie'
  812 = 'C2- ciecie'
  537 = 'C2- podawanie'
  70 = 'Ciecie 1'
  806 = 'Ciecie 2'
  0 = 'Clear'
  436 = 'Data koniec'
  435 = 'Data start'
  376 = 'DO ZROBIENIA :\n- Wysyłanie komunikatów od maszyny\n- Poprawienie wizualizacji logowanie błędów\n\n\n\n\n\n- Użytkownicy ograniczenia w dodawanych modulach\n\n\n- Języki tłumaczenia'
  475 = 'DO ZROBIENIA :\n- Wysyłanie komunikatów od maszyny\n- Poprawienie wizualizacji logowanie błędów\n-Użytkownicy całość\n\n\n\n\n\n\n- Języki tłumaczenia'
  46 = 'Filtr'
  936 = 'Hold'
  432 = 'Kod'
  922 = 'Login'
  63 = 'Logout'
  579 = 'None'
  431 = 'Nr Elem.'
  384 = 'Operator'
  434 = 'Opis'
  410 = 'Ostzreżenia'
  707 = 'Podaj'
  687 = 'Podawanie - bazowanie'
  564 = 'Podawanie - podawanie'
  973 = 'Podawanie wafla'
  433 = 'R'
  573 = 'Reset'
  188 = 'Service'
  125 = 'Start'
  387 = 'Stop'
  986 = 'Suspend'
  332 = 'Test jezykow - Domyslny'
  892 = 'Tryb automatyczny'
  732 = 'Tryb półautomatyczny'
  740 = 'Tryb reczny'
  916 = 'Tylko aktywne'
  974 = 'Un-hold'
  152 = 'Un-Suspend'
  13 = 'User: %s'
  460 = 'Wafel do C1'
  762 = 'Wafel do C2'
  374 = 'Wafel do podania'
  528 = 'Wiadomości'
  609 = 'Zmiana hasła'
  411 = 'Zmien'
END_TEXTLIST

// ---- POUs/90 - Stan Maszyny/Visu/Visu_StanMaszyny_AktualyStan.TcVIS
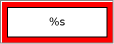
VISUALIZATION Visu_StanMaszyny_AktualyStan  // 114x44
VAR_IN_OUT
	bNacisniety								: BOOL;
END_VAR
VAR_INPUT
	stVisuStan								: DUT_StanMaszyny_VISU_Stan;
END_VAR
    RoundedRectangle (2,2 110x40), invisible if: not stVisuStan.bAktywny
    RoundedRectangle (7,7 100x30), "%s", text variable: stVisuStan.sNazwa, colour variable: 16#FF000000 OR (16#FF000000 OR (stVisuStan.dwKolorTla))
        OnMouseDown: execute {
            //IF (stVisuStan.bAktywny) THEN
            	bNacisniety := stVisuStan.bAktywny AND TRUE;
            //END_IF
        }
END_VISUALIZATION

// ---- POUs/90 - Stan Maszyny/Visu/Visu_StanMaszyny_AktualyStan_BezNaciskania.TcVIS
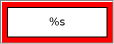
VISUALIZATION Visu_StanMaszyny_AktualyStan_BezNaciskania  // 114x44
VAR_IN_OUT
	
END_VAR
VAR_INPUT
	stVisuStan								: DUT_StanMaszyny_VISU_Stan;
END_VAR
    RoundedRectangle (2,2 110x40), invisible if: not stVisuStan.bAktywny
    RoundedRectangle (7,7 100x30), "%s", text variable: stVisuStan.sNazwa, colour variable: 16#FF000000 OR (16#FF000000 OR (stVisuStan.dwKolorTla))
END_VISUALIZATION

// ---- POUs/90 - Stan Maszyny/Visu/Visu_StanMaszyny_Diagram.TcVIS
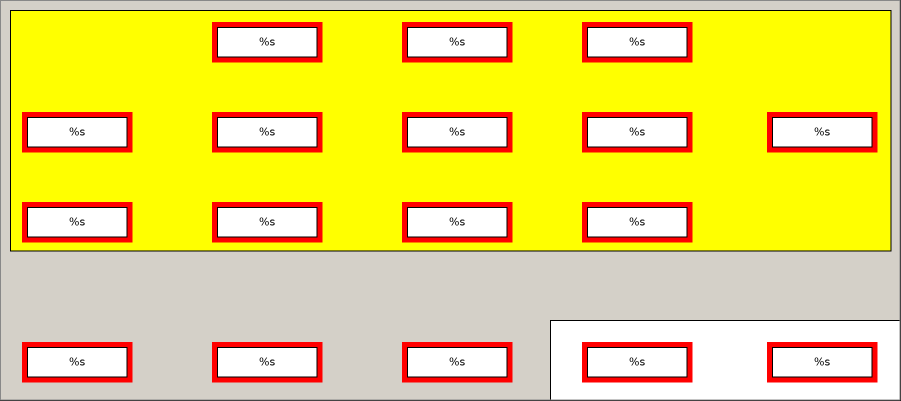
VISUALIZATION Visu_StanMaszyny_Diagram  // 901x401
VAR_IN_OUT
	
